LIN {X 0,Y 324.452,Z 606.51,A -85,B 0,C 180,E1 -15849.821,E2 -15849.821} C_VEL
LIN {X 0,Y 327.125,Z 593.397,A -85,B 0,C 180,E1 -15851.148,E2 -15851.148} C_VEL
LIN {X 0,Y 329.681,Z 579.293,A -85,B 0,C 180,E1 -15852.308,E2 -15852.308} C_VEL
LIN {X 0,Y 332.153,Z 563.092,A -85,B 0,C 180,E1 -15853.333,E2 -15853.333} C_VEL
LIN {X 0,Y 333.966,Z 548.09,A -85,B 0,C 180,E1 -15854.029,E2 -15854.029} C_VEL
LIN {X 0,Y 336.479,Z 518.568,A -85,B 0,C 180,E1 -15854.979,E2 -15854.979} C_VEL
LIN {X 0,Y 343.808,Z 437.667,A -85,B 0,C 180,E1 -15857.456,E2 -15857.456} C_VEL
LIN {X 0,Y 343.461,Z 436.268,A -85,B 0,C 180,E1 -15857.604,E2 -15857.604} C_VEL
LIN {X 0,Y 340.27,Z 429.347,A -85,B 0,C 180,E1 -15858.7,E2 -15858.7} C_VEL
LIN {X 0,Y 336.483,Z 422.195,A -85,B 0,C 180,E1 -15860.082,E2 -15860.082} C_VEL
LIN {X 0,Y 332.788,Z 415.874,A -85,B 0,C 180,E1 -15861.56,E2 -15861.56} C_VEL
LIN {X 0,Y 329.389,Z 410.762,A -85,B 0,C 180,E1 -15863.052,E2 -15863.052} C_VEL
LIN {X 0,Y 326.443,Z 406.618,A -85,B 0,C 180,E1 -15864.518,E2 -15864.518} C_VEL
LIN {X 0,Y 322.983,Z 401.962,A -85,B 0,C 180,E1 -15866.589,E2 -15866.589} C_VEL
LIN {X 0,Y 319.205,Z 397.297,A -85,B 0,C 180,E1 -15869.678,E2 -15869.678} C_VEL
LIN {X 0,Y 316.987,Z 395.124,A -85,B 0,C 180,E1 -15872.902,E2 -15872.902} C_VEL
LIN {X 0,Y 316.478,Z 394.789,A -85,B 0,C 180,E1 -15875.266,E2 -15875.266} C_VEL
LIN {X 0,Y 316.828,Z 395.766,A -85,B 0,C 180,E1 -15877.528,E2 -15877.528} C_VEL
LIN {X 0,Y 318.754,Z 398.698,A -85,B 0,C 180,E1 -15880.662,E2 -15880.662} C_VEL
LIN {X 0,Y 320.871,Z 401.495,A -85,B 0,C 180,E1 -15882.648,E2 -15882.648} C_VEL
LIN {X 0,Y 325.084,Z 407.921,A -85,B 0,C 180,E1 -15885.514,E2 -15885.514} C_VEL
LIN {X 0,Y 328.982,Z 414.436,A -85,B 0,C 180,E1 -15887.591,E2 -15887.591} C_VEL
LIN {X 0,Y 332.395,Z 420.455,A -85,B 0,C 180,E1 -15889.134,E2 -15889.134} C_VEL
LIN {X 0,Y 336.259,Z 427.81,A -85,B 0,C 180,E1 -15890.698,E2 -15890.698} C_VEL
LIN {X 0,Y 340.531,Z 437.373,A -85,B 0,C 180,E1 -15892.295,E2 -15892.295} C_VEL
LIN {X 0,Y 342.927,Z 443.986,A -85,B 0,C 180,E1 -15893.182,E2 -15893.182} C_VEL
LIN {X 0,Y 343.146,Z 448.361,A -85,B 0,C 180,E1 -15893.458,E2 -15893.458} C_VEL
LIN {X 0,Y 334.823,Z 544.074,A -85,B 0,C 180,E1 -15896.383,E2 -15896.383} C_VEL
LIN {X 0,Y 333.156,Z 562.468,A -85,B 0,C 180,E1 -15897.006,E2 -15897.006} C_VEL
LIN {X 0,Y 330.94,Z 578.482,A -85,B 0,C 180,E1 -15897.752,E2 -15897.752} C_VEL
LIN {X 0,Y 328.466,Z 592.922,A -85,B 0,C 180,E1 -15898.653,E2 -15898.653} C_VEL
LIN {X 0,Y 325.617,Z 607.581,A -85,B 0,C 180,E1 -15899.828,E2 -15899.828} C_VEL
LIN {X 0,Y 322.66,Z 621.222,A -85,B 0,C 180,E1 -15901.188,E2 -15901.188} C_VEL
LIN {X 0,Y 319.496,Z 634.657,A -85,B 0,C 180,E1 -15902.841,E2 -15902.841} C_VEL
LIN {X 0,Y 316.461,Z 646.925,A -85,B 0,C 180,E1 -15904.689,E2 -15904.689} C_VEL
LIN {X 0,Y 313.386,Z 658.797,A -85,B 0,C 180,E1 -15906.848,E2 -15906.848} C_VEL
LIN {X 0,Y 310.733,Z 669.029,A -85,B 0,C 180,E1 -15909.13,E2 -15909.13} C_VEL
LIN {X 0,Y 308.293,Z 678.544,A -85,B 0,C 180,E1 -15911.731,E2 -15911.731} C_VEL
LIN {X 0,Y 306.546,Z 685.471,A -85,B 0,C 180,E1 -15914.029,E2 -15914.029} C_VEL
LIN {X 0,Y 305.238,Z 691.852,A -85,B 0,C 180,E1 -15916.687,E2 -15916.687} C_VEL
LIN {X 0,Y 304.288,Z 696.815,A -85,B 0,C 180,E1 -15919.35,E2 -15919.35} C_VEL
LIN {X 0,Y 303.795,Z 700.457,A -85,B 0,C 180,E1 -15922.019,E2 -15922.019} C_VEL
LIN {X 0,Y 303.596,Z 702.832,A -85,B 0,C 180,E1 -15924.685,E2 -15924.685} C_VEL
LIN {X 0,Y 303.593,Z 703.983,A -85,B 0,C 180,E1 -15927.344,E2 -15927.344} C_VEL
LIN {X 0,Y 303.605,Z 703.898,A -85,B 0,C 180,E1 -15929.998,E2 -15929.998} C_VEL
LIN {X 0,Y 303.619,Z 702.551,A -85,B 0,C 180,E1 -15932.651,E2 -15932.651} C_VEL
LIN {X 0,Y 303.634,Z 699.89,A -85,B 0,C 180,E1 -15935.31,E2 -15935.31} C_VEL
LIN {X 0,Y 303.805,Z 695.853,A -85,B 0,C 180,E1 -15937.976,E2 -15937.976} C_VEL
LIN {X 0,Y 304.12,Z 690.347,A -85,B 0,C 180,E1 -15940.652,E2 -15940.652} C_VEL
LIN {X 0,Y 304.708,Z 685.156,A -85,B 0,C 180,E1 -15942.655,E2 -15942.655} C_VEL
LIN {X 0,Y 305.549,Z 677.938,A -85,B 0,C 180,E1 -15944.973,E2 -15944.973} C_VEL
LIN {X 0,Y 306.797,Z 669.033,A -85,B 0,C 180,E1 -15947.323,E2 -15947.323} C_VEL
LIN {X 0,Y 308.202,Z 660.042,A -85,B 0,C 180,E1 -15949.306,E2 -15949.306} C_VEL
LIN {X 0,Y 309.836,Z 649.388,A -85,B 0,C 180,E1 -15951.278,E2 -15951.278} C_VEL
LIN {X 0,Y 311.797,Z 636.624,A -85,B 0,C 180,E1 -15953.23,E2 -15953.23} C_VEL
LIN {X 0,Y 313.659,Z 623.857,A -85,B 0,C 180,E1 -15954.84,E2 -15954.84} C_VEL
LIN {X 0,Y 315.546,Z 609.954,A -85,B 0,C 180,E1 -15956.272,E2 -15956.272} C_VEL
LIN {X 0,Y 317.457,Z 594.626,A -85,B 0,C 180,E1 -15957.523,E2 -15957.523} C_VEL
LIN {X 0,Y 319.021,Z 579.208,A -85,B 0,C 180,E1 -15958.492,E2 -15958.492} C_VEL
LIN {X 0,Y 320.355,Z 563.283,A -85,B 0,C 180,E1 -15959.215,E2 -15959.215} C_VEL
LIN {X 0,Y 321.454,Z 541.44,A -85,B 0,C 180,E1 -15959.87,E2 -15959.87} C_VEL
LIN {X 0,Y 325.806,Z 442.848,A -85,B 0,C 180,E1 -15962.583,E2 -15962.583} C_VEL
LIN {X 0,Y 322.744,Z 425.216,A -85,B 0,C 180,E1 -15963.398,E2 -15963.398} C_VEL
LIN {X 0,Y 310.834,Z 396.248,A -85,B 0,C 180,E1 -15965.467,E2 -15965.467} C_VEL
LIN {X 0,Y 309.569,Z 393.101,A -85,B 0,C 180,E1 -15965.719,E2 -15965.719} C_VEL
LIN {X 0,Y 306.644,Z 381.762,A -85,B 0,C 180,E1 -15968.809,E2 -15968.809} C_VEL
LIN {X 0,Y 305.41,Z 377.069,A -85,B 0,C 180,E1 -15970.171,E2 -15970.171} C_VEL
LIN {X 0,Y 305.411,Z 377.066,A -85,B 0,C 180,E1 -15973.654,E2 -15973.654} C_VEL
LIN {X 0,Y 305.424,Z 377.063,A -85,B 0,C 180,E1 -15977.417,E2 -15977.417} C_VEL
LIN {X 0,Y 305.429,Z 377.064,A -85,B 0,C 180,E1 -15981.591,E2 -15981.591} C_VEL
LIN {X 0,Y 305.449,Z 377.06,A -85,B 0,C 180,E1 -15984.885,E2 -15984.885} C_VEL
LIN {X 0,Y 305.429,Z 377.065,A -85,B 0,C 180,E1 -15988.357,E2 -15988.357} C_VEL
LIN {X 0,Y 305.44,Z 377.06,A -85,B 0,C 180,E1 -15991.106,E2 -15991.106} C_VEL
LIN {X 0,Y 305.465,Z 377.06,A -85,B 0,C 180,E1 -15994.079,E2 -15994.079} C_VEL
LIN {X 0,Y 305.447,Z 377.062,A -85,B 0,C 180,E1 -15998.399,E2 -15998.399} C_VEL
LIN {X 0,Y 305.5,Z 377.049,A -85,B 0,C 180,E1 -16001.212,E2 -16001.212} C_VEL
LIN {X 0,Y 305.566,Z 377.045,A -85,B 0,C 180,E1 -16005.345,E2 -16005.345} C_VEL
LIN {X 0,Y 305.609,Z 377.036,A -85,B 0,C 180,E1 -16009.399,E2 -16009.399} C_VEL
LIN {X 0,Y 305.732,Z 377.027,A -85,B 0,C 180,E1 -16012.073,E2 -16012.073} C_VEL
LIN {X 0,Y 305.643,Z 377.035,A -85,B 0,C 180,E1 -16014.723,E2 -16014.723} C_VEL
LIN {X 0,Y 305.92,Z 377.001,A -85,B 0,C 180,E1 -16018.684,E2 -16018.684} C_VEL
LIN {X 0,Y 305.92,Z 377.001,A -85,B 0,C 180,E1 -16021.317,E2 -16021.317} C_VEL
LIN {X 0,Y 305.771,Z 377.02,A -85,B 0,C 180,E1 -16026.6,E2 -16026.6} C_VEL
LIN {X 0,Y 305.68,Z 377.03,A -85,B 0,C 180,E1 -16029.262,E2 -16029.262} C_VEL
LIN {X 0,Y 305.556,Z 377.046,A -85,B 0,C 180,E1 -16033.298,E2 -16033.298} C_VEL
LIN {X 0,Y 305.51,Z 377.051,A -85,B 0,C 180,E1 -16037.401,E2 -16037.401} C_VEL
LIN {X 0,Y 305.468,Z 377.06,A -85,B 0,C 180,E1 -16040.189,E2 -16040.189} C_VEL
LIN {X 0,Y 305.442,Z 377.059,A -85,B 0,C 180,E1 -16044.467,E2 -16044.467} C_VEL
LIN {X 0,Y 305.429,Z 377.061,A -85,B 0,C 180,E1 -16047.401,E2 -16047.401} C_VEL
LIN {X 0,Y 305.406,Z 377.065,A -85,B 0,C 180,E1 -16050.416,E2 -16050.416} C_VEL
LIN {X 0,Y 305.454,Z 377.06,A -85,B 0,C 180,E1 -16054.08,E2 -16054.08} C_VEL
LIN {X 0,Y 305.441,Z 377.059,A -85,B 0,C 180,E1 -16056.745,E2 -16056.745} C_VEL
LIN {X 0,Y 305.4,Z 377.064,A -85,B 0,C 180,E1 -16060.592,E2 -16060.592} C_VEL
LIN {X 0,Y 305.413,Z 377.065,A -85,B 0,C 180,E1 -16063.658,E2 -16063.658} C_VEL
LIN {X 0,Y 305.427,Z 377.064,A -85,B 0,C 180,E1 -16067.421,E2 -16067.421} C_VEL
LIN {X 0,Y 305.435,Z 377.062,A -85,B 0,C 180,E1 -16071.594,E2 -16071.594} C_VEL
LIN {X 0,Y 305.455,Z 377.058,A -85,B 0,C 180,E1 -16074.889,E2 -16074.889} C_VEL
LIN {X 0,Y 305.437,Z 377.06,A -85,B 0,C 180,E1 -16078.361,E2 -16078.361} C_VEL
LIN {X 0,Y 305.45,Z 377.059,A -85,B 0,C 180,E1 -16081.109,E2 -16081.109} C_VEL
LIN {X 0,Y 305.476,Z 377.057,A -85,B 0,C 180,E1 -16084.082,E2 -16084.082} C_VEL
LIN {X 0,Y 305.463,Z 377.058,A -85,B 0,C 180,E1 -16088.403,E2 -16088.403} C_VEL
LIN {X 0,Y 305.542,Z 377.048,A -85,B 0,C 180,E1 -16091.217,E2 -16091.217} C_VEL
LIN {X 0,Y 305.626,Z 377.032,A -85,B 0,C 180,E1 -16095.35,E2 -16095.35} C_VEL
LIN {X 0,Y 305.636,Z 377.038,A -85,B 0,C 180,E1 -16099.402,E2 -16099.402} C_VEL
LIN {X 0,Y 305.747,Z 377.023,A -85,B 0,C 180,E1 -16102.075,E2 -16102.075} C_VEL
LIN {X 0,Y 305.659,Z 377.029,A -85,B 0,C 180,E1 -16104.725,E2 -16104.725} C_VEL
LIN {X 0,Y 305.948,Z 376.997,A -85,B 0,C 180,E1 -16108.686,E2 -16108.686} C_VEL
LIN {X 0,Y 305.939,Z 377.001,A -85,B 0,C 180,E1 -16111.318,E2 -16111.318} C_VEL
LIN {X 0,Y 305.664,Z 377.035,A -85,B 0,C 180,E1 -16115.279,E2 -16115.279} C_VEL
LIN {X 0,Y 305.763,Z 377.022,A -85,B 0,C 180,E1 -16117.929,E2 -16117.929} C_VEL
LIN {X 0,Y 305.6,Z 377.043,A -85,B 0,C 180,E1 -16121.947,E2 -16121.947} C_VEL
LIN {X 0,Y 305.564,Z 377.044,A -85,B 0,C 180,E1 -16124.981,E2 -16124.981} C_VEL
LIN {X 0,Y 305.515,Z 377.05,A -85,B 0,C 180,E1 -16128.789,E2 -16128.789} C_VEL
LIN {X 0,Y 305.492,Z 377.055,A -85,B 0,C 180,E1 -16133.041,E2 -16133.041} C_VEL
LIN {X 0,Y 305.459,Z 377.059,A -85,B 0,C 180,E1 -16136.192,E2 -16136.192} C_VEL
LIN {X 0,Y 305.455,Z 377.061,A -85,B 0,C 180,E1 -16139.035,E2 -16139.035} C_VEL
LIN {X 0,Y 305.443,Z 377.064,A -85,B 0,C 180,E1 -16141.954,E2 -16141.954} C_VEL
LIN {X 0,Y 305.515,Z 377.213,A -85,B 0,C 180,E1 -16145.029,E2 -16145.029} C_VEL
LIN {X 0,Y 306.526,Z 379.933,A -85,B 0,C 180,E1 -16145.226,E2 -16145.226} C_VEL
LIN {X 0,Y 311.318,Z 389.798,A -85,B 0,C 180,E1 -16146.039,E2 -16146.039} C_VEL
LIN {X 0,Y 322.35,Z 415.707,A -85,B 0,C 180,E1 -16147.921,E2 -16147.921} C_VEL
LIN {X 0,Y 326.082,Z 424.987,A -85,B 0,C 180,E1 -16148.538,E2 -16148.538} C_VEL
LIN {X 0,Y 320.68,Z 542.492,A -85,B 0,C 180,E1 -16151.776,E2 -16151.776} C_VEL
LIN {X 0,Y 319.54,Z 558.615,A -85,B 0,C 180,E1 -16152.473,E2 -16152.473} C_VEL
LIN {X 0,Y 318.124,Z 574.349,A -85,B 0,C 180,E1 -16153.424,E2 -16153.424} C_VEL
LIN {X 0,Y 316.452,Z 589.23,A -85,B 0,C 180,E1 -16154.596,E2 -16154.596} C_VEL
LIN {X 0,Y 314.644,Z 603.29,A -85,B 0,C 180,E1 -16155.985,E2 -16155.985} C_VEL
LIN {X 0,Y 312.776,Z 616.701,A -85,B 0,C 180,E1 -16157.616,E2 -16157.616} C_VEL
LIN {X 0,Y 310.867,Z 629.385,A -85,B 0,C 180,E1 -16159.492,E2 -16159.492} C_VEL
LIN {X 0,Y 309.241,Z 639.693,A -85,B 0,C 180,E1 -16161.319,E2 -16161.319} C_VEL
LIN {X 0,Y 307.978,Z 647.89,A -85,B 0,C 180,E1 -16163.009,E2 -16163.009} C_VEL
LIN {X 0,Y 306.745,Z 651.603,A -85,B 0,C 180,E1 -16163.849,E2 -16163.849} C_VEL
LIN {X 0,Y 303.068,Z 657.329,A -85,B 0,C 180,E1 -16165.212,E2 -16165.212} C_VEL
LIN {X 0,Y 299.488,Z 662.573,A -85,B 0,C 180,E1 -16166.655,E2 -16166.655} C_VEL
LIN {X 0,Y 298.416,Z 665.551,A -85,B 0,C 180,E1 -16167.604,E2 -16167.604} C_VEL
LIN {X 0,Y 297.562,Z 672.589,A -85,B 0,C 180,E1 -16170.264,E2 -16170.264} C_VEL
LIN {X 0,Y 297.025,Z 677.318,A -85,B 0,C 180,E1 -16172.522,E2 -16172.522} C_VEL
LIN {X 0,Y 296.632,Z 681.037,A -85,B 0,C 180,E1 -16174.756,E2 -16174.756} C_VEL
LIN {X 0,Y 296.351,Z 684.552,A -85,B 0,C 180,E1 -16177.7,E2 -16177.7} C_VEL
LIN {X 0,Y 296.213,Z 686.564,A -85,B 0,C 180,E1 -16180.599,E2 -16180.599} C_VEL
LIN {X 0,Y 296.266,Z 687.043,A -85,B 0,C 180,E1 -16182.038,E2 -16182.038} C_VEL
LIN {X 0,Y 296.413,Z 686.992,A -85,B 0,C 180,E1 -16184.881,E2 -16184.881} C_VEL
LIN {X 0,Y 296.859,Z 685.634,A -85,B 0,C 180,E1 -16187.697,E2 -16187.697} C_VEL
LIN {X 0,Y 297.577,Z 683.019,A -85,B 0,C 180,E1 -16190.484,E2 -16190.484} C_VEL
LIN {X 0,Y 298.656,Z 679.093,A -85,B 0,C 180,E1 -16193.243,E2 -16193.243} C_VEL
LIN {X 0,Y 300.16,Z 673.803,A -85,B 0,C 180,E1 -16195.972,E2 -16195.972} C_VEL
LIN {X 0,Y 302.276,Z 666.695,A -85,B 0,C 180,E1 -16198.809,E2 -16198.809} C_VEL
LIN {X 0,Y 304.679,Z 658.733,A -85,B 0,C 180,E1 -16201.321,E2 -16201.321} C_VEL
LIN {X 0,Y 307.304,Z 649.837,A -85,B 0,C 180,E1 -16203.605,E2 -16203.605} C_VEL
LIN {X 0,Y 310.461,Z 639.239,A -85,B 0,C 180,E1 -16205.847,E2 -16205.847} C_VEL
LIN {X 0,Y 313.734,Z 627.426,A -85,B 0,C 180,E1 -16207.886,E2 -16207.886} C_VEL
LIN {X 0,Y 317.103,Z 614.32,A -85,B 0,C 180,E1 -16209.729,E2 -16209.729} C_VEL
LIN {X 0,Y 320.152,Z 601.331,A -85,B 0,C 180,E1 -16211.234,E2 -16211.234} C_VEL
LIN {X 0,Y 323.061,Z 587.136,A -85,B 0,C 180,E1 -16212.564,E2 -16212.564} C_VEL
LIN {X 0,Y 325.711,Z 572.302,A -85,B 0,C 180,E1 -16213.651,E2 -16213.651} C_VEL
LIN {X 0,Y 327.75,Z 558.503,A -85,B 0,C 180,E1 -16214.453,E2 -16214.453} C_VEL
LIN {X 0,Y 329.623,Z 542.223,A -85,B 0,C 180,E1 -16215.14,E2 -16215.14} C_VEL
LIN {X 0,Y 339.186,Z 441.013,A -85,B 0,C 180,E1 -16218.308,E2 -16218.308} C_VEL
LIN {X 0,Y 339.127,Z 439.74,A -85,B 0,C 180,E1 -16218.392,E2 -16218.392} C_VEL
LIN {X 0,Y 335.275,Z 431.44,A -85,B 0,C 180,E1 -16219.832,E2 -16219.832} C_VEL
LIN {X 0,Y 331.155,Z 423.968,A -85,B 0,C 180,E1 -16221.494,E2 -16221.494} C_VEL
LIN {X 0,Y 327.497,Z 417.79,A -85,B 0,C 180,E1 -16223.175,E2 -16223.175} C_VEL
LIN {X 0,Y 324.214,Z 413.03,A -85,B 0,C 180,E1 -16224.882,E2 -16224.882} C_VEL
LIN {X 0,Y 321.15,Z 408.709,A -85,B 0,C 180,E1 -16226.809,E2 -16226.809} C_VEL
LIN {X 0,Y 317.586,Z 404.164,A -85,B 0,C 180,E1 -16229.844,E2 -16229.844} C_VEL
LIN {X 0,Y 315.511,Z 402.045,A -85,B 0,C 180,E1 -16232.995,E2 -16232.995} C_VEL
LIN {X 0,Y 315.041,Z 401.783,A -85,B 0,C 180,E1 -16235.451,E2 -16235.451} C_VEL
LIN {X 0,Y 315.502,Z 402.97,A -85,B 0,C 180,E1 -16237.839,E2 -16237.839} C_VEL
LIN {X 0,Y 317.445,Z 406.025,A -85,B 0,C 180,E1 -16240.865,E2 -16240.865} C_VEL
LIN {X 0,Y 319.074,Z 408.27,A -85,B 0,C 180,E1 -16242.403,E2 -16242.403} C_VEL
LIN {X 0,Y 322.847,Z 414.322,A -85,B 0,C 180,E1 -16245.135,E2 -16245.135} C_VEL
LIN {X 0,Y 326.288,Z 420.329,A -85,B 0,C 180,E1 -16247.082,E2 -16247.082} C_VEL
LIN {X 0,Y 329.432,Z 426.175,A -85,B 0,C 180,E1 -16248.617,E2 -16248.617} C_VEL
LIN {X 0,Y 333.083,Z 433.543,A -85,B 0,C 180,E1 -16250.207,E2 -16250.207} C_VEL
LIN {X 0,Y 337.359,Z 443.689,A -85,B 0,C 180,E1 -16251.915,E2 -16251.915} C_VEL
LIN {X 0,Y 338.627,Z 447.338,A -85,B 0,C 180,E1 -16252.402,E2 -16252.402} C_VEL
LIN {X 0,Y 338.62,Z 450.838,A -85,B 0,C 180,E1 -16252.588,E2 -16252.588} C_VEL
LIN {X 0,Y 330.386,Z 539.529,A -85,B 0,C 180,E1 -16255.362,E2 -16255.362} C_VEL
LIN {X 0,Y 328.263,Z 561.131,A -85,B 0,C 180,E1 -16256.081,E2 -16256.081} C_VEL
LIN {X 0,Y 325.98,Z 577.135,A -85,B 0,C 180,E1 -16256.832,E2 -16256.832} C_VEL
LIN {X 0,Y 323.342,Z 591.833,A -85,B 0,C 180,E1 -16257.73,E2 -16257.73} C_VEL
LIN {X 0,Y 320.323,Z 606.661,A -85,B 0,C 180,E1 -16258.916,E2 -16258.916} C_VEL
LIN {X 0,Y 316.915,Z 621.573,A -85,B 0,C 180,E1 -16260.432,E2 -16260.432} C_VEL
LIN {X 0,Y 313.295,Z 635.94,A -85,B 0,C 180,E1 -16262.257,E2 -16262.257} C_VEL
LIN {X 0,Y 310.126,Z 647.958,A -85,B 0,C 180,E1 -16264.134,E2 -16264.134} C_VEL
LIN {X 0,Y 307.304,Z 658.157,A -85,B 0,C 180,E1 -16266.045,E2 -16266.045} C_VEL
LIN {X 0,Y 304.467,Z 668.311,A -85,B 0,C 180,E1 -16268.324,E2 -16268.324} C_VEL
LIN {X 0,Y 302.122,Z 676.804,A -85,B 0,C 180,E1 -16270.639,E2 -16270.639} C_VEL
LIN {X 0,Y 300.204,Z 683.887,A -85,B 0,C 180,E1 -16272.982,E2 -16272.982} C_VEL
LIN {X 0,Y 298.827,Z 689.05,A -85,B 0,C 180,E1 -16275.005,E2 -16275.005} C_VEL
LIN {X 0,Y 297.701,Z 694.624,A -85,B 0,C 180,E1 -16277.731,E2 -16277.731} C_VEL
LIN {X 0,Y 296.951,Z 698.826,A -85,B 0,C 180,E1 -16280.462,E2 -16280.462} C_VEL
LIN {X 0,Y 296.554,Z 701.735,A -85,B 0,C 180,E1 -16283.193,E2 -16283.193} C_VEL
LIN {X 0,Y 296.467,Z 703.408,A -85,B 0,C 180,E1 -16285.92,E2 -16285.92} C_VEL
LIN {X 0,Y 296.491,Z 703.855,A -85,B 0,C 180,E1 -16288.64,E2 -16288.64} C_VEL
LIN {X 0,Y 296.512,Z 703.056,A -85,B 0,C 180,E1 -16291.356,E2 -16291.356} C_VEL
LIN {X 0,Y 296.551,Z 700.983,A -85,B 0,C 180,E1 -16294.075,E2 -16294.075} C_VEL
LIN {X 0,Y 296.629,Z 697.572,A -85,B 0,C 180,E1 -16296.801,E2 -16296.801} C_VEL
LIN {X 0,Y 296.882,Z 692.722,A -85,B 0,C 180,E1 -16299.536,E2 -16299.536} C_VEL
LIN {X 0,Y 297.49,Z 686.32,A -85,B 0,C 180,E1 -16302.274,E2 -16302.274} C_VEL
LIN {X 0,Y 298.239,Z 679.294,A -85,B 0,C 180,E1 -16304.672,E2 -16304.672} C_VEL
LIN {X 0,Y 299.517,Z 670.79,A -85,B 0,C 180,E1 -16307.054,E2 -16307.054} C_VEL
LIN {X 0,Y 301.118,Z 660.526,A -85,B 0,C 180,E1 -16309.424,E2 -16309.424} C_VEL
LIN {X 0,Y 302.819,Z 649.975,A -85,B 0,C 180,E1 -16311.438,E2 -16311.438} C_VEL
LIN {X 0,Y 304.586,Z 638.51,A -85,B 0,C 180,E1 -16313.272,E2 -16313.272} C_VEL
LIN {X 0,Y 306.497,Z 626.146,A -85,B 0,C 180,E1 -16314.917,E2 -16314.917} C_VEL
LIN {X 0,Y 308.403,Z 612.791,A -85,B 0,C 180,E1 -16316.381,E2 -16316.381} C_VEL
LIN {X 0,Y 310.342,Z 598.348,A -85,B 0,C 180,E1 -16317.654,E2 -16317.654} C_VEL
LIN {X 0,Y 311.967,Z 582.868,A -85,B 0,C 180,E1 -16318.728,E2 -16318.728} C_VEL
LIN {X 0,Y 313.407,Z 567.509,A -85,B 0,C 180,E1 -16319.507,E2 -16319.507} C_VEL
LIN {X 0,Y 314.469,Z 550.42,A -85,B 0,C 180,E1 -16320.093,E2 -16320.093} C_VEL
LIN {X 0,Y 319.42,Z 444.085,A -85,B 0,C 180,E1 -16323.081,E2 -16323.081} C_VEL
LIN {X 0,Y 316.595,Z 427.87,A -85,B 0,C 180,E1 -16323.856,E2 -16323.856} C_VEL
LIN {X 0,Y 305.243,Z 399.983,A -85,B 0,C 180,E1 -16325.887,E2 -16325.887} C_VEL
LIN {X 0,Y 302.268,Z 392.932,A -85,B 0,C 180,E1 -16326.455,E2 -16326.455} C_VEL
LIN {X 0,Y 299.308,Z 381.624,A -85,B 0,C 180,E1 -16329.63,E2 -16329.63} C_VEL
LIN {X 0,Y 298.352,Z 377.947,A -85,B 0,C 180,E1 -16330.708,E2 -16330.708} C_VEL
LIN {X 0,Y 298.36,Z 377.944,A -85,B 0,C 180,E1 -16333.096,E2 -16333.096} C_VEL
LIN {X 0,Y 298.36,Z 377.944,A -85,B 0,C 180,E1 -16336.913,E2 -16336.913} C_VEL
LIN {X 0,Y 298.373,Z 377.942,A -85,B 0,C 180,E1 -16341.01,E2 -16341.01} C_VEL
LIN {X 0,Y 298.392,Z 377.943,A -85,B 0,C 180,E1 -16343.927,E2 -16343.927} C_VEL
LIN {X 0,Y 298.38,Z 377.941,A -85,B 0,C 180,E1 -16347.198,E2 -16347.198} C_VEL
LIN {X 0,Y 298.351,Z 377.945,A -85,B 0,C 180,E1 -16350.637,E2 -16350.637} C_VEL
LIN {X 0,Y 298.407,Z 377.935,A -85,B 0,C 180,E1 -16354.917,E2 -16354.917} C_VEL
LIN {X 0,Y 298.403,Z 377.937,A -85,B 0,C 180,E1 -16359.312,E2 -16359.312} C_VEL
LIN {X 0,Y 298.445,Z 377.934,A -85,B 0,C 180,E1 -16362.174,E2 -16362.174} C_VEL
LIN {X 0,Y 298.498,Z 377.925,A -85,B 0,C 180,E1 -16364.99,E2 -16364.99} C_VEL
LIN {X 0,Y 298.568,Z 377.912,A -85,B 0,C 180,E1 -16369.146,E2 -16369.146} C_VEL
LIN {X 0,Y 298.684,Z 377.903,A -85,B 0,C 180,E1 -16371.884,E2 -16371.884} C_VEL
LIN {X 0,Y 298.613,Z 377.912,A -85,B 0,C 180,E1 -16374.598,E2 -16374.598} C_VEL
LIN {X 0,Y 298.888,Z 377.877,A -85,B 0,C 180,E1 -16378.653,E2 -16378.653} C_VEL
LIN {X 0,Y 298.888,Z 377.877,A -85,B 0,C 180,E1 -16381.348,E2 -16381.348} C_VEL
LIN {X 0,Y 298.72,Z 377.898,A -85,B 0,C 180,E1 -16386.756,E2 -16386.756} C_VEL
LIN {X 0,Y 298.611,Z 377.911,A -85,B 0,C 180,E1 -16389.483,E2 -16389.483} C_VEL
LIN {X 0,Y 298.509,Z 377.926,A -85,B 0,C 180,E1 -16393.618,E2 -16393.618} C_VEL
LIN {X 0,Y 298.446,Z 377.931,A -85,B 0,C 180,E1 -16396.415,E2 -16396.415} C_VEL
LIN {X 0,Y 298.427,Z 377.935,A -85,B 0,C 180,E1 -16399.617,E2 -16399.617} C_VEL
LIN {X 0,Y 298.376,Z 377.942,A -85,B 0,C 180,E1 -16403.605,E2 -16403.605} C_VEL
LIN {X 0,Y 298.389,Z 377.937,A -85,B 0,C 180,E1 -16406.584,E2 -16406.584} C_VEL
LIN {X 0,Y 298.346,Z 377.947,A -85,B 0,C 180,E1 -16409.65,E2 -16409.65} C_VEL
LIN {X 0,Y 298.382,Z 377.938,A -85,B 0,C 180,E1 -16412.802,E2 -16412.802} C_VEL
LIN {X 0,Y 298.416,Z 377.934,A -85,B 0,C 180,E1 -16416.804,E2 -16416.804} C_VEL
LIN {X 0,Y 298.364,Z 377.944,A -85,B 0,C 180,E1 -16419.494,E2 -16419.494} C_VEL
LIN {X 0,Y 298.362,Z 377.939,A -85,B 0,C 180,E1 -16423.099,E2 -16423.099} C_VEL
LIN {X 0,Y 298.363,Z 377.942,A -85,B 0,C 180,E1 -16426.917,E2 -16426.917} C_VEL
LIN {X 0,Y 298.344,Z 377.941,A -85,B 0,C 180,E1 -16431.021,E2 -16431.021} C_VEL
LIN {X 0,Y 298.398,Z 377.942,A -85,B 0,C 180,E1 -16433.93,E2 -16433.93} C_VEL
LIN {X 0,Y 298.388,Z 377.939,A -85,B 0,C 180,E1 -16437.202,E2 -16437.202} C_VEL
LIN {X 0,Y 298.36,Z 377.942,A -85,B 0,C 180,E1 -16440.64,E2 -16440.64} C_VEL
LIN {X 0,Y 298.418,Z 377.934,A -85,B 0,C 180,E1 -16444.921,E2 -16444.921} C_VEL
LIN {X 0,Y 298.4,Z 377.942,A -85,B 0,C 180,E1 -16447.865,E2 -16447.865} C_VEL
LIN {X 0,Y 298.502,Z 377.924,A -85,B 0,C 180,E1 -16450.757,E2 -16450.757} C_VEL
LIN {X 0,Y 298.586,Z 377.906,A -85,B 0,C 180,E1 -16454.997,E2 -16454.997} C_VEL
LIN {X 0,Y 298.592,Z 377.914,A -85,B 0,C 180,E1 -16459.149,E2 -16459.149} C_VEL
LIN {X 0,Y 298.699,Z 377.902,A -85,B 0,C 180,E1 -16461.886,E2 -16461.886} C_VEL
LIN {X 0,Y 298.629,Z 377.904,A -85,B 0,C 180,E1 -16464.6,E2 -16464.6} C_VEL
LIN {X 0,Y 298.915,Z 377.874,A -85,B 0,C 180,E1 -16468.655,E2 -16468.655} C_VEL
LIN {X 0,Y 298.906,Z 377.877,A -85,B 0,C 180,E1 -16471.349,E2 -16471.349} C_VEL
LIN {X 0,Y 298.744,Z 377.896,A -85,B 0,C 180,E1 -16476.757,E2 -16476.757} C_VEL
LIN {X 0,Y 298.63,Z 377.911,A -85,B 0,C 180,E1 -16479.484,E2 -16479.484} C_VEL
LIN {X 0,Y 298.529,Z 377.924,A -85,B 0,C 180,E1 -16483.618,E2 -16483.618} C_VEL
LIN {X 0,Y 298.46,Z 377.93,A -85,B 0,C 180,E1 -16486.416,E2 -16486.416} C_VEL
LIN {X 0,Y 298.464,Z 377.934,A -85,B 0,C 180,E1 -16489.628,E2 -16489.628} C_VEL
LIN {X 0,Y 298.422,Z 377.94,A -85,B 0,C 180,E1 -16493.603,E2 -16493.603} C_VEL
LIN {X 0,Y 298.409,Z 377.937,A -85,B 0,C 180,E1 -16496.584,E2 -16496.584} C_VEL
LIN {X 0,Y 298.4,Z 377.942,A -85,B 0,C 180,E1 -16499.645,E2 -16499.645} C_VEL
LIN {X 0,Y 298.442,Z 377.937,A -85,B 0,C 180,E1 -16504.009,E2 -16504.009} C_VEL
LIN {X 0,Y 298.437,Z 377.936,A -85,B 0,C 180,E1 -16504.315,E2 -16504.315} C_VEL
LIN {X 0,Y 299.471,Z 380.811,A -85,B 0,C 180,E1 -16504.536,E2 -16504.536} C_VEL
LIN {X 0,Y 305.256,Z 392.555,A -85,B 0,C 180,E1 -16505.547,E2 -16505.547} C_VEL
LIN {X 0,Y 316.025,Z 417.81,A -85,B 0,C 180,E1 -16507.425,E2 -16507.425} C_VEL
LIN {X 0,Y 319.644,Z 426.763,A -85,B 0,C 180,E1 -16508.04,E2 -16508.04} C_VEL
LIN {X 0,Y 314.082,Z 542.928,A -85,B 0,C 180,E1 -16511.322,E2 -16511.322} C_VEL
LIN {X 0,Y 312.92,Z 558.734,A -85,B 0,C 180,E1 -16512.019,E2 -16512.019} C_VEL
LIN {X 0,Y 311.501,Z 574.104,A -85,B 0,C 180,E1 -16512.963,E2 -16512.963} C_VEL
LIN {X 0,Y 309.761,Z 589.124,A -85,B 0,C 180,E1 -16514.162,E2 -16514.162} C_VEL
LIN {X 0,Y 307.816,Z 603.741,A -85,B 0,C 180,E1 -16515.635,E2 -16515.635} C_VEL
LIN {X 0,Y 305.858,Z 617.372,A -85,B 0,C 180,E1 -16517.334,E2 -16517.334} C_VEL
LIN {X 0,Y 303.949,Z 629.768,A -85,B 0,C 180,E1 -16519.216,E2 -16519.216} C_VEL
LIN {X 0,Y 302.258,Z 640.203,A -85,B 0,C 180,E1 -16521.112,E2 -16521.112} C_VEL
LIN {X 0,Y 300.611,Z 650.718,A -85,B 0,C 180,E1 -16523.404,E2 -16523.404} C_VEL
LIN {X 0,Y 299.259,Z 659.412,A -85,B 0,C 180,E1 -16525.692,E2 -16525.692} C_VEL
LIN {X 0,Y 298.416,Z 665.551,A -85,B 0,C 180,E1 -16527.604,E2 -16527.604} C_VEL
LIN {X 0,Y 297.377,Z 668.411,A -85,B 0,C 180,E1 -16528.578,E2 -16528.578} C_VEL
LIN {X 0,Y 293.991,Z 672.622,A -85,B 0,C 180,E1 -16530.191,E2 -16530.191} C_VEL
LIN {X 0,Y 290.711,Z 676.311,A -85,B 0,C 180,E1 -16531.887,E2 -16531.887} C_VEL
LIN {X 0,Y 289.862,Z 678.327,A -85,B 0,C 180,E1 -16532.975,E2 -16532.975} C_VEL
LIN {X 0,Y 289.384,Z 682.358,A -85,B 0,C 180,E1 -16535.615,E2 -16535.615} C_VEL
LIN {X 0,Y 289.26,Z 684.409,A -85,B 0,C 180,E1 -16537.412,E2 -16537.412} C_VEL
LIN {X 0,Y 289.133,Z 686.47,A -85,B 0,C 180,E1 -16540.104,E2 -16540.104} C_VEL
LIN {X 0,Y 289.19,Z 687.4,A -85,B 0,C 180,E1 -16543.044,E2 -16543.044} C_VEL
LIN {X 0,Y 289.516,Z 686.916,A -85,B 0,C 180,E1 -16546.173,E2 -16546.173} C_VEL
LIN {X 0,Y 290.01,Z 685.293,A -85,B 0,C 180,E1 -16548.821,E2 -16548.821} C_VEL
LIN {X 0,Y 291.035,Z 681.984,A -85,B 0,C 180,E1 -16551.932,E2 -16551.932} C_VEL
LIN {X 0,Y 292.188,Z 678.07,A -85,B 0,C 180,E1 -16554.479,E2 -16554.479} C_VEL
LIN {X 0,Y 293.983,Z 672.461,A -85,B 0,C 180,E1 -16557.259,E2 -16557.259} C_VEL
LIN {X 0,Y 296.247,Z 665.349,A -85,B 0,C 180,E1 -16560,E2 -16560} C_VEL
LIN {X 0,Y 299.086,Z 656.561,A -85,B 0,C 180,E1 -16562.693,E2 -16562.693} C_VEL
LIN {X 0,Y 302.085,Z 647.247,A -85,B 0,C 180,E1 -16565.005,E2 -16565.005} C_VEL
LIN {X 0,Y 305.474,Z 636.234,A -85,B 0,C 180,E1 -16567.234,E2 -16567.234} C_VEL
LIN {X 0,Y 308.843,Z 624.704,A -85,B 0,C 180,E1 -16569.165,E2 -16569.165} C_VEL
LIN {X 0,Y 312.156,Z 612.34,A -85,B 0,C 180,E1 -16570.868,E2 -16570.868} C_VEL
LIN {X 0,Y 315.459,Z 598.809,A -85,B 0,C 180,E1 -16572.382,E2 -16572.382} C_VEL
LIN {X 0,Y 318.168,Z 586.129,A -85,B 0,C 180,E1 -16573.557,E2 -16573.557} C_VEL
LIN {X 0,Y 321.001,Z 570.965,A -85,B 0,C 180,E1 -16574.665,E2 -16574.665} C_VEL
LIN {X 0,Y 323.31,Z 555.555,A -85,B 0,C 180,E1 -16575.524,E2 -16575.524} C_VEL
LIN {X 0,Y 325.279,Z 538.493,A -85,B 0,C 180,E1 -16576.191,E2 -16576.191} C_VEL
LIN {X 0,Y 334.765,Z 444.063,A -85,B 0,C 180,E1 -16579.206,E2 -16579.206} C_VEL
LIN {X 0,Y 334.731,Z 442.837,A -85,B 0,C 180,E1 -16579.287,E2 -16579.287} C_VEL
LIN {X 0,Y 330.67,Z 434.216,A -85,B 0,C 180,E1 -16580.933,E2 -16580.933} C_VEL
LIN {X 0,Y 326.849,Z 427.251,A -85,B 0,C 180,E1 -16582.646,E2 -16582.646} C_VEL
LIN {X 0,Y 324.275,Z 423.039,A -85,B 0,C 180,E1 -16583.936,E2 -16583.936} C_VEL
LIN {X 0,Y 321.87,Z 419.311,A -85,B 0,C 180,E1 -16585.314,E2 -16585.314} C_VEL
LIN {X 0,Y 319.167,Z 415.297,A -85,B 0,C 180,E1 -16587.136,E2 -16587.136} C_VEL
LIN {X 0,Y 315.978,Z 411.027,A -85,B 0,C 180,E1 -16590.012,E2 -16590.012} C_VEL
LIN {X 0,Y 314,Z 408.924,A -85,B 0,C 180,E1 -16593.174,E2 -16593.174} C_VEL
LIN {X 0,Y 313.656,Z 408.808,A -85,B 0,C 180,E1 -16595.929,E2 -16595.929} C_VEL
LIN {X 0,Y 314.451,Z 410.753,A -85,B 0,C 180,E1 -16598.741,E2 -16598.741} C_VEL
LIN {X 0,Y 316.851,Z 414.176,A -85,B 0,C 180,E1 -16601.714,E2 -16601.714} C_VEL
LIN {X 0,Y 320.66,Z 420.804,A -85,B 0,C 180,E1 -16604.774,E2 -16604.774} C_VEL
LIN {X 0,Y 323.864,Z 426.734,A -85,B 0,C 180,E1 -16606.707,E2 -16606.707} C_VEL
LIN {X 0,Y 326.571,Z 431.988,A -85,B 0,C 180,E1 -16608.111,E2 -16608.111} C_VEL
LIN {X 0,Y 329.931,Z 439.147,A -85,B 0,C 180,E1 -16609.668,E2 -16609.668} C_VEL
LIN {X 0,Y 333.796,Z 448.773,A -85,B 0,C 180,E1 -16611.318,E2 -16611.318} C_VEL
LIN {X 0,Y 334.441,Z 450.771,A -85,B 0,C 180,E1 -16611.603,E2 -16611.603} C_VEL
LIN {X 0,Y 323.578,Z 559.492,A -85,B 0,C 180,E1 -16615.096,E2 -16615.096} C_VEL
LIN {X 0,Y 321.137,Z 576.408,A -85,B 0,C 180,E1 -16615.887,E2 -16615.887} C_VEL
LIN {X 0,Y 318.18,Z 592.007,A -85,B 0,C 180,E1 -16616.859,E2 -16616.859} C_VEL
LIN {X 0,Y 314.95,Z 606.819,A -85,B 0,C 180,E1 -16618.072,E2 -16618.072} C_VEL
LIN {X 0,Y 311.614,Z 620.769,A -85,B 0,C 180,E1 -16619.504,E2 -16619.504} C_VEL
LIN {X 0,Y 308.127,Z 634.068,A -85,B 0,C 180,E1 -16621.193,E2 -16621.193} C_VEL
LIN {X 0,Y 304.987,Z 645.262,A -85,B 0,C 180,E1 -16622.926,E2 -16622.926} C_VEL
LIN {X 0,Y 301.874,Z 655.828,A -85,B 0,C 180,E1 -16624.855,E2 -16624.855} C_VEL
LIN {X 0,Y 299.077,Z 664.879,A -85,B 0,C 180,E1 -16626.819,E2 -16626.819} C_VEL
LIN {X 0,Y 296.414,Z 673.846,A -85,B 0,C 180,E1 -16629.165,E2 -16629.165} C_VEL
LIN {X 0,Y 294.535,Z 680.426,A -85,B 0,C 180,E1 -16631.206,E2 -16631.206} C_VEL
LIN {X 0,Y 292.383,Z 687.579,A -85,B 0,C 180,E1 -16633.895,E2 -16633.895} C_VEL
LIN {X 0,Y 291.05,Z 693.482,A -85,B 0,C 180,E1 -16636.736,E2 -16636.736} C_VEL
LIN {X 0,Y 290.223,Z 696.951,A -85,B 0,C 180,E1 -16638.828,E2 -16638.828} C_VEL
LIN {X 0,Y 289.664,Z 700.433,A -85,B 0,C 180,E1 -16641.627,E2 -16641.627} C_VEL
LIN {X 0,Y 289.427,Z 702.742,A -85,B 0,C 180,E1 -16644.609,E2 -16644.609} C_VEL
LIN {X 0,Y 289.419,Z 703.593,A -85,B 0,C 180,E1 -16647.214,E2 -16647.214} C_VEL
LIN {X 0,Y 289.438,Z 703.326,A -85,B 0,C 180,E1 -16649.998,E2 -16649.998} C_VEL
LIN {X 0,Y 289.471,Z 701.796,A -85,B 0,C 180,E1 -16652.781,E2 -16652.781} C_VEL
LIN {X 0,Y 289.499,Z 698.958,A -85,B 0,C 180,E1 -16655.57,E2 -16655.57} C_VEL
LIN {X 0,Y 289.68,Z 694.738,A -85,B 0,C 180,E1 -16658.368,E2 -16658.368} C_VEL
LIN {X 0,Y 290.047,Z 689.008,A -85,B 0,C 180,E1 -16661.175,E2 -16661.175} C_VEL
LIN {X 0,Y 290.822,Z 682.687,A -85,B 0,C 180,E1 -16663.626,E2 -16663.626} C_VEL
LIN {X 0,Y 291.88,Z 674.925,A -85,B 0,C 180,E1 -16666.073,E2 -16666.073} C_VEL
LIN {X 0,Y 293.256,Z 665.539,A -85,B 0,C 180,E1 -16668.512,E2 -16668.512} C_VEL
LIN {X 0,Y 294.87,Z 655.932,A -85,B 0,C 180,E1 -16670.58,E2 -16670.58} C_VEL
LIN {X 0,Y 296.645,Z 644.754,A -85,B 0,C 180,E1 -16672.603,E2 -16672.603} C_VEL
LIN {X 0,Y 298.525,Z 633.332,A -85,B 0,C 180,E1 -16674.328,E2 -16674.328} C_VEL
LIN {X 0,Y 300.592,Z 619.993,A -85,B 0,C 180,E1 -16675.998,E2 -16675.998} C_VEL
LIN {X 0,Y 302.632,Z 605.349,A -85,B 0,C 180,E1 -16677.485,E2 -16677.485} C_VEL
LIN {X 0,Y 304.557,Z 590.331,A -85,B 0,C 180,E1 -16678.683,E2 -16678.683} C_VEL
LIN {X 0,Y 306.081,Z 575.704,A -85,B 0,C 180,E1 -16679.579,E2 -16679.579} C_VEL
LIN {X 0,Y 307.379,Z 559.601,A -85,B 0,C 180,E1 -16680.292,E2 -16680.292} C_VEL
LIN {X 0,Y 312.947,Z 444.922,A -85,B 0,C 180,E1 -16683.622,E2 -16683.622} C_VEL
LIN {X 0,Y 310.521,Z 430.46,A -85,B 0,C 180,E1 -16684.331,E2 -16684.331} C_VEL
LIN {X 0,Y 298.148,Z 400.247,A -85,B 0,C 180,E1 -16686.588,E2 -16686.588} C_VEL
LIN {X 0,Y 294.969,Z 392.699,A -85,B 0,C 180,E1 -16687.231,E2 -16687.231} C_VEL
LIN {X 0,Y 291.301,Z 378.825,A -85,B 0,C 180,E1 -16691.325,E2 -16691.325} C_VEL
LIN {X 0,Y 291.271,Z 378.827,A -85,B 0,C 180,E1 -16695.595,E2 -16695.595} C_VEL
LIN {X 0,Y 291.288,Z 378.825,A -85,B 0,C 180,E1 -16699.35,E2 -16699.35} C_VEL
LIN {X 0,Y 291.373,Z 378.814,A -85,B 0,C 180,E1 -16702.915,E2 -16702.915} C_VEL
LIN {X 0,Y 291.331,Z 378.823,A -85,B 0,C 180,E1 -16706.3,E2 -16706.3} C_VEL
LIN {X 0,Y 291.322,Z 378.823,A -85,B 0,C 180,E1 -16710.277,E2 -16710.277} C_VEL
LIN {X 0,Y 291.332,Z 378.819,A -85,B 0,C 180,E1 -16714.264,E2 -16714.264} C_VEL
LIN {X 0,Y 291.337,Z 378.818,A -85,B 0,C 180,E1 -16717.296,E2 -16717.296} C_VEL
LIN {X 0,Y 291.373,Z 378.812,A -85,B 0,C 180,E1 -16720.265,E2 -16720.265} C_VEL
LIN {X 0,Y 291.46,Z 378.803,A -85,B 0,C 180,E1 -16724.682,E2 -16724.682} C_VEL
LIN {X 0,Y 291.513,Z 378.79,A -85,B 0,C 180,E1 -16728.88,E2 -16728.88} C_VEL
LIN {X 0,Y 291.637,Z 378.779,A -85,B 0,C 180,E1 -16731.687,E2 -16731.687} C_VEL
LIN {X 0,Y 291.583,Z 378.788,A -85,B 0,C 180,E1 -16734.468,E2 -16734.468} C_VEL
LIN {X 0,Y 291.856,Z 378.753,A -85,B 0,C 180,E1 -16738.621,E2 -16738.621} C_VEL
LIN {X 0,Y 291.855,Z 378.753,A -85,B 0,C 180,E1 -16741.38,E2 -16741.38} C_VEL
LIN {X 0,Y 291.673,Z 378.775,A -85,B 0,C 180,E1 -16746.92,E2 -16746.92} C_VEL
LIN {X 0,Y 291.554,Z 378.792,A -85,B 0,C 180,E1 -16749.715,E2 -16749.715} C_VEL
LIN {X 0,Y 291.468,Z 378.806,A -85,B 0,C 180,E1 -16753.953,E2 -16753.953} C_VEL
LIN {X 0,Y 291.382,Z 378.812,A -85,B 0,C 180,E1 -16758.274,E2 -16758.274} C_VEL
LIN {X 0,Y 291.332,Z 378.818,A -85,B 0,C 180,E1 -16761.215,E2 -16761.215} C_VEL
LIN {X 0,Y 291.321,Z 378.819,A -85,B 0,C 180,E1 -16764.213,E2 -16764.213} C_VEL
LIN {X 0,Y 291.317,Z 378.818,A -85,B 0,C 180,E1 -16767.283,E2 -16767.283} C_VEL
LIN {X 0,Y 291.291,Z 378.824,A -85,B 0,C 180,E1 -16770.443,E2 -16770.443} C_VEL
LIN {X 0,Y 291.333,Z 378.819,A -85,B 0,C 180,E1 -16773.7,E2 -16773.7} C_VEL
LIN {X 0,Y 291.342,Z 378.816,A -85,B 0,C 180,E1 -16777.25,E2 -16777.25} C_VEL
LIN {X 0,Y 291.291,Z 378.821,A -85,B 0,C 180,E1 -16780.65,E2 -16780.65} C_VEL
LIN {X 0,Y 291.274,Z 378.825,A -85,B 0,C 180,E1 -16784.406,E2 -16784.406} C_VEL
LIN {X 0,Y 291.287,Z 378.823,A -85,B 0,C 180,E1 -16788.414,E2 -16788.414} C_VEL
LIN {X 0,Y 291.379,Z 378.811,A -85,B 0,C 180,E1 -16792.918,E2 -16792.918} C_VEL
LIN {X 0,Y 291.338,Z 378.817,A -85,B 0,C 180,E1 -16796.304,E2 -16796.304} C_VEL
LIN {X 0,Y 291.331,Z 378.819,A -85,B 0,C 180,E1 -16800.281,E2 -16800.281} C_VEL
LIN {X 0,Y 291.343,Z 378.816,A -85,B 0,C 180,E1 -16804.268,E2 -16804.268} C_VEL
LIN {X 0,Y 291.357,Z 378.815,A -85,B 0,C 180,E1 -16807.3,E2 -16807.3} C_VEL
LIN {X 0,Y 291.438,Z 378.805,A -85,B 0,C 180,E1 -16810.271,E2 -16810.271} C_VEL
LIN {X 0,Y 291.497,Z 378.787,A -85,B 0,C 180,E1 -16814.668,E2 -16814.668} C_VEL
LIN {X 0,Y 291.536,Z 378.792,A -85,B 0,C 180,E1 -16818.883,E2 -16818.883} C_VEL
LIN {X 0,Y 291.653,Z 378.782,A -85,B 0,C 180,E1 -16821.689,E2 -16821.689} C_VEL
LIN {X 0,Y 291.599,Z 378.779,A -85,B 0,C 180,E1 -16824.47,E2 -16824.47} C_VEL
LIN {X 0,Y 291.881,Z 378.75,A -85,B 0,C 180,E1 -16828.622,E2 -16828.622} C_VEL
LIN {X 0,Y 291.874,Z 378.753,A -85,B 0,C 180,E1 -16831.382,E2 -16831.382} C_VEL
LIN {X 0,Y 291.696,Z 378.774,A -85,B 0,C 180,E1 -16836.921,E2 -16836.921} C_VEL
LIN {X 0,Y 291.573,Z 378.79,A -85,B 0,C 180,E1 -16839.716,E2 -16839.716} C_VEL
LIN {X 0,Y 291.487,Z 378.799,A -85,B 0,C 180,E1 -16843.954,E2 -16843.954} C_VEL
LIN {X 0,Y 291.398,Z 378.809,A -85,B 0,C 180,E1 -16848.274,E2 -16848.274} C_VEL
LIN {X 0,Y 291.366,Z 378.817,A -85,B 0,C 180,E1 -16851.214,E2 -16851.214} C_VEL
LIN {X 0,Y 291.356,Z 378.816,A -85,B 0,C 180,E1 -16854.211,E2 -16854.211} C_VEL
LIN {X 0,Y 291.357,Z 378.818,A -85,B 0,C 180,E1 -16857.28,E2 -16857.28} C_VEL
LIN {X 0,Y 291.325,Z 378.821,A -85,B 0,C 180,E1 -16860.44,E2 -16860.44} C_VEL
LIN {X 0,Y 291.414,Z 378.834,A -85,B 0,C 180,E1 -16863.602,E2 -16863.602} C_VEL
LIN {X 0,Y 292.397,Z 381.656,A -85,B 0,C 180,E1 -16863.814,E2 -16863.814} C_VEL
LIN {X 0,Y 299.127,Z 395.138,A -85,B 0,C 180,E1 -16865.023,E2 -16865.023} C_VEL
LIN {X 0,Y 309.326,Z 418.968,A -85,B 0,C 180,E1 -16866.843,E2 -16866.843} C_VEL
LIN {X 0,Y 313.243,Z 428.722,A -85,B 0,C 180,E1 -16867.531,E2 -16867.531} C_VEL
LIN {X 0,Y 307.483,Z 543.32,A -85,B 0,C 180,E1 -16870.851,E2 -16870.851} C_VEL
LIN {X 0,Y 306.285,Z 559.008,A -85,B 0,C 180,E1 -16871.562,E2 -16871.562} C_VEL
LIN {X 0,Y 304.891,Z 573.582,A -85,B 0,C 180,E1 -16872.47,E2 -16872.47} C_VEL
LIN {X 0,Y 303.292,Z 587.71,A -85,B 0,C 180,E1 -16873.602,E2 -16873.602} C_VEL
LIN {X 0,Y 301.466,Z 600.996,A -85,B 0,C 180,E1 -16874.917,E2 -16874.917} C_VEL
LIN {X 0,Y 299.564,Z 614.169,A -85,B 0,C 180,E1 -16876.517,E2 -16876.517} C_VEL
LIN {X 0,Y 297.547,Z 626.745,A -85,B 0,C 180,E1 -16878.37,E2 -16878.37} C_VEL
LIN {X 0,Y 295.911,Z 636.668,A -85,B 0,C 180,E1 -16880.114,E2 -16880.114} C_VEL
LIN {X 0,Y 294.094,Z 647.86,A -85,B 0,C 180,E1 -16882.455,E2 -16882.455} C_VEL
LIN {X 0,Y 292.639,Z 657.096,A -85,B 0,C 180,E1 -16884.803,E2 -16884.803} C_VEL
LIN {X 0,Y 291.298,Z 666.101,A -85,B 0,C 180,E1 -16887.613,E2 -16887.613} C_VEL
LIN {X 0,Y 290.499,Z 672.569,A -85,B 0,C 180,E1 -16890.116,E2 -16890.116} C_VEL
LIN {X 0,Y 289.862,Z 678.327,A -85,B 0,C 180,E1 -16892.975,E2 -16892.975} C_VEL
LIN {X 0,Y 289.029,Z 680.185,A -85,B 0,C 180,E1 -16894.073,E2 -16894.073} C_VEL
LIN {X 0,Y 285.881,Z 682.761,A -85,B 0,C 180,E1 -16895.876,E2 -16895.876} C_VEL
LIN {X 0,Y 283.266,Z 684.451,A -85,B 0,C 180,E1 -16897.362,E2 -16897.362} C_VEL
LIN {X 0,Y 282.134,Z 685.483,A -85,B 0,C 180,E1 -16898.528,E2 -16898.528} C_VEL
LIN {X 0,Y 282.033,Z 685.74,A -85,B 0,C 180,E1 -16898.926,E2 -16898.926} C_VEL
LIN {X 0,Y 282.044,Z 687.107,A -85,B 0,C 180,E1 -16901.247,E2 -16901.247} C_VEL
LIN {X 0,Y 282.141,Z 687.637,A -85,B 0,C 180,E1 -16904.097,E2 -16904.097} C_VEL
LIN {X 0,Y 282.551,Z 686.908,A -85,B 0,C 180,E1 -16907.064,E2 -16907.064} C_VEL
LIN {X 0,Y 283.257,Z 684.906,A -85,B 0,C 180,E1 -16909.998,E2 -16909.998} C_VEL
LIN {X 0,Y 284.368,Z 681.651,A -85,B 0,C 180,E1 -16912.901,E2 -16912.901} C_VEL
LIN {X 0,Y 285.898,Z 677.074,A -85,B 0,C 180,E1 -16915.77,E2 -16915.77} C_VEL
LIN {X 0,Y 287.966,Z 671.089,A -85,B 0,C 180,E1 -16918.601,E2 -16918.601} C_VEL
LIN {X 0,Y 290.53,Z 663.649,A -85,B 0,C 180,E1 -16921.386,E2 -16921.386} C_VEL
LIN {X 0,Y 293.379,Z 655.624,A -85,B 0,C 180,E1 -16923.777,E2 -16923.777} C_VEL
LIN {X 0,Y 296.666,Z 645.835,A -85,B 0,C 180,E1 -16926.188,E2 -16926.188} C_VEL
LIN {X 0,Y 300.304,Z 634.762,A -85,B 0,C 180,E1 -16928.41,E2 -16928.41} C_VEL
LIN {X 0,Y 304.199,Z 621.971,A -85,B 0,C 180,E1 -16930.482,E2 -16930.482} C_VEL
LIN {X 0,Y 307.803,Z 609.112,A -85,B 0,C 180,E1 -16932.193,E2 -16932.193} C_VEL
LIN {X 0,Y 311.166,Z 595.688,A -85,B 0,C 180,E1 -16933.643,E2 -16933.643} C_VEL
LIN {X 0,Y 314.018,Z 582.388,A -85,B 0,C 180,E1 -16934.816,E2 -16934.816} C_VEL
LIN {X 0,Y 317.033,Z 566.25,A -85,B 0,C 180,E1 -16935.922,E2 -16935.922} C_VEL
LIN {X 0,Y 319.362,Z 550.788,A -85,B 0,C 180,E1 -16936.706,E2 -16936.706} C_VEL
LIN {X 0,Y 321.522,Z 530.982,A -85,B 0,C 180,E1 -16937.409,E2 -16937.409} C_VEL
LIN {X 0,Y 330.566,Z 446.377,A -85,B 0,C 180,E1 -16940.165,E2 -16940.165} C_VEL
LIN {X 0,Y 327.135,Z 438.934,A -85,B 0,C 180,E1 -16941.683,E2 -16941.683} C_VEL
LIN {X 0,Y 323.809,Z 432.663,A -85,B 0,C 180,E1 -16943.305,E2 -16943.305} C_VEL
LIN {X 0,Y 321.544,Z 428.77,A -85,B 0,C 180,E1 -16944.537,E2 -16944.537} C_VEL
LIN {X 0,Y 319.323,Z 425.294,A -85,B 0,C 180,E1 -16945.879,E2 -16945.879} C_VEL
LIN {X 0,Y 317.06,Z 421.744,A -85,B 0,C 180,E1 -16947.543,E2 -16947.543} C_VEL
LIN {X 0,Y 314.372,Z 417.887,A -85,B 0,C 180,E1 -16950.181,E2 -16950.181} C_VEL
LIN {X 0,Y 312.491,Z 415.809,A -85,B 0,C 180,E1 -16953.355,E2 -16953.355} C_VEL
LIN {X 0,Y 312.23,Z 415.901,A -85,B 0,C 180,E1 -16956.119,E2 -16956.119} C_VEL
LIN {X 0,Y 313.039,Z 417.834,A -85,B 0,C 180,E1 -16958.818,E2 -16958.818} C_VEL
LIN {X 0,Y 315.181,Z 421.09,A -85,B 0,C 180,E1 -16961.556,E2 -16961.556} C_VEL
LIN {X 0,Y 318.499,Z 427.226,A -85,B 0,C 180,E1 -16964.386,E2 -16964.386} C_VEL
LIN {X 0,Y 321.299,Z 432.715,A -85,B 0,C 180,E1 -16966.206,E2 -16966.206} C_VEL
LIN {X 0,Y 324.118,Z 438.551,A -85,B 0,C 180,E1 -16967.762,E2 -16967.762} C_VEL
LIN {X 0,Y 327.228,Z 445.717,A -85,B 0,C 180,E1 -16969.303,E2 -16969.303} C_VEL
LIN {X 0,Y 330.159,Z 453.574,A -85,B 0,C 180,E1 -16970.666,E2 -16970.666} C_VEL
LIN {X 0,Y 320.515,Z 545.513,A -85,B 0,C 180,E1 -16973.648,E2 -16973.648} C_VEL
LIN {X 0,Y 318.447,Z 563.342,A -85,B 0,C 180,E1 -16974.304,E2 -16974.304} C_VEL
LIN {X 0,Y 315.718,Z 579.583,A -85,B 0,C 180,E1 -16975.121,E2 -16975.121} C_VEL
LIN {X 0,Y 312.421,Z 595.596,A -85,B 0,C 180,E1 -16976.205,E2 -16976.205} C_VEL
LIN {X 0,Y 309.174,Z 609.393,A -85,B 0,C 180,E1 -16977.403,E2 -16977.403} C_VEL
LIN {X 0,Y 305.667,Z 622.72,A -85,B 0,C 180,E1 -16978.845,E2 -16978.845} C_VEL
LIN {X 0,Y 301.703,Z 636.634,A -85,B 0,C 180,E1 -16980.711,E2 -16980.711} C_VEL
LIN {X 0,Y 298.187,Z 648.369,A -85,B 0,C 180,E1 -16982.637,E2 -16982.637} C_VEL
LIN {X 0,Y 295.006,Z 658.38,A -85,B 0,C 180,E1 -16984.606,E2 -16984.606} C_VEL
LIN {X 0,Y 291.795,Z 668.346,A -85,B 0,C 180,E1 -16986.957,E2 -16986.957} C_VEL
LIN {X 0,Y 289.138,Z 676.731,A -85,B 0,C 180,E1 -16989.361,E2 -16989.361} C_VEL
LIN {X 0,Y 286.61,Z 684.648,A -85,B 0,C 180,E1 -16992.149,E2 -16992.149} C_VEL
LIN {X 0,Y 284.673,Z 691.041,A -85,B 0,C 180,E1 -16994.974,E2 -16994.974} C_VEL
LIN {X 0,Y 283.491,Z 695.994,A -85,B 0,C 180,E1 -16997.833,E2 -16997.833} C_VEL
LIN {X 0,Y 282.861,Z 698.859,A -85,B 0,C 180,E1 -16999.982,E2 -16999.982} C_VEL
LIN {X 0,Y 282.396,Z 701.621,A -85,B 0,C 180,E1 -17002.85,E2 -17002.85} C_VEL
LIN {X 0,Y 282.283,Z 703.118,A -85,B 0,C 180,E1 -17005.714,E2 -17005.714} C_VEL
LIN {X 0,Y 282.335,Z 703.374,A -85,B 0,C 180,E1 -17008.572,E2 -17008.572} C_VEL
LIN {X 0,Y 282.355,Z 702.383,A -85,B 0,C 180,E1 -17011.424,E2 -17011.424} C_VEL
LIN {X 0,Y 282.399,Z 701.41,A -85,B 0,C 180,E1 -17012.851,E2 -17012.851} C_VEL
LIN {X 0,Y 282.409,Z 698.463,A -85,B 0,C 180,E1 -17015.711,E2 -17015.711} C_VEL
LIN {X 0,Y 282.605,Z 694.126,A -85,B 0,C 180,E1 -17018.579,E2 -17018.579} C_VEL
LIN {X 0,Y 283.019,Z 688.267,A -85,B 0,C 180,E1 -17021.456,E2 -17021.456} C_VEL
LIN {X 0,Y 283.842,Z 681.811,A -85,B 0,C 180,E1 -17023.968,E2 -17023.968} C_VEL
LIN {X 0,Y 284.935,Z 673.918,A -85,B 0,C 180,E1 -17026.476,E2 -17026.476} C_VEL
LIN {X 0,Y 286.414,Z 664.347,A -85,B 0,C 180,E1 -17028.971,E2 -17028.971} C_VEL
LIN {X 0,Y 288.087,Z 654.589,A -85,B 0,C 180,E1 -17031.087,E2 -17031.087} C_VEL
LIN {X 0,Y 290.01,Z 642.978,A -85,B 0,C 180,E1 -17033.188,E2 -17033.188} C_VEL
LIN {X 0,Y 292.136,Z 630.258,A -85,B 0,C 180,E1 -17035.085,E2 -17035.085} C_VEL
LIN {X 0,Y 294.318,Z 616.265,A -85,B 0,C 180,E1 -17036.787,E2 -17036.787} C_VEL
LIN {X 0,Y 296.289,Z 602.681,A -85,B 0,C 180,E1 -17038.125,E2 -17038.125} C_VEL
LIN {X 0,Y 298.109,Z 588.017,A -85,B 0,C 180,E1 -17039.275,E2 -17039.275} C_VEL
LIN {X 0,Y 299.688,Z 572.899,A -85,B 0,C 180,E1 -17040.178,E2 -17040.178} C_VEL
LIN {X 0,Y 300.916,Z 556.68,A -85,B 0,C 180,E1 -17040.867,E2 -17040.867} C_VEL
LIN {X 0,Y 306.559,Z 446.079,A -85,B 0,C 180,E1 -17044.16,E2 -17044.16} C_VEL
LIN {X 0,Y 304.328,Z 432.908,A -85,B 0,C 180,E1 -17044.817,E2 -17044.817} C_VEL
LIN {X 0,Y 292.355,Z 403.525,A -85,B 0,C 180,E1 -17047.074,E2 -17047.074} C_VEL
LIN {X 0,Y 287.62,Z 392.468,A -85,B 0,C 180,E1 -17048.048,E2 -17048.048} C_VEL
LIN {X 0,Y 284.244,Z 379.704,A -85,B 0,C 180,E1 -17051.938,E2 -17051.938} C_VEL
LIN {X 0,Y 284.227,Z 379.707,A -85,B 0,C 180,E1 -17056.184,E2 -17056.184} C_VEL
LIN {X 0,Y 284.272,Z 379.702,A -85,B 0,C 180,E1 -17060.028,E2 -17060.028} C_VEL
LIN {X 0,Y 284.306,Z 379.696,A -85,B 0,C 180,E1 -17063.611,E2 -17063.611} C_VEL
LIN {X 0,Y 284.294,Z 379.696,A -85,B 0,C 180,E1 -17067.189,E2 -17067.189} C_VEL
LIN {X 0,Y 284.296,Z 379.697,A -85,B 0,C 180,E1 -17070.369,E2 -17070.369} C_VEL
LIN {X 0,Y 284.283,Z 379.696,A -85,B 0,C 180,E1 -17073.577,E2 -17073.577} C_VEL
LIN {X 0,Y 284.296,Z 379.696,A -85,B 0,C 180,E1 -17076.701,E2 -17076.701} C_VEL
LIN {X 0,Y 284.32,Z 379.693,A -85,B 0,C 180,E1 -17079.927,E2 -17079.927} C_VEL
LIN {X 0,Y 284.418,Z 379.681,A -85,B 0,C 180,E1 -17084.503,E2 -17084.503} C_VEL
LIN {X 0,Y 284.445,Z 379.671,A -85,B 0,C 180,E1 -17088.6,E2 -17088.6} C_VEL
LIN {X 0,Y 284.594,Z 379.654,A -85,B 0,C 180,E1 -17091.48,E2 -17091.48} C_VEL
LIN {X 0,Y 284.553,Z 379.665,A -85,B 0,C 180,E1 -17094.331,E2 -17094.331} C_VEL
LIN {X 0,Y 284.823,Z 379.629,A -85,B 0,C 180,E1 -17098.586,E2 -17098.586} C_VEL
LIN {X 0,Y 284.823,Z 379.63,A -85,B 0,C 180,E1 -17101.414,E2 -17101.414} C_VEL
LIN {X 0,Y 284.628,Z 379.653,A -85,B 0,C 180,E1 -17107.092,E2 -17107.092} C_VEL
LIN {X 0,Y 284.5,Z 379.67,A -85,B 0,C 180,E1 -17109.958,E2 -17109.958} C_VEL
LIN {X 0,Y 284.405,Z 379.683,A -85,B 0,C 180,E1 -17114.307,E2 -17114.307} C_VEL
LIN {X 0,Y 284.344,Z 379.686,A -85,B 0,C 180,E1 -17117.254,E2 -17117.254} C_VEL
LIN {X 0,Y 284.31,Z 379.695,A -85,B 0,C 180,E1 -17120.248,E2 -17120.248} C_VEL
LIN {X 0,Y 284.286,Z 379.699,A -85,B 0,C 180,E1 -17123.844,E2 -17123.844} C_VEL
LIN {X 0,Y 284.274,Z 379.695,A -85,B 0,C 180,E1 -17127.131,E2 -17127.131} C_VEL
LIN {X 0,Y 284.263,Z 379.701,A -85,B 0,C 180,E1 -17130.086,E2 -17130.086} C_VEL
LIN {X 0,Y 284.294,Z 379.692,A -85,B 0,C 180,E1 -17132.947,E2 -17132.947} C_VEL
LIN {X 0,Y 284.308,Z 379.693,A -85,B 0,C 180,E1 -17136.39,E2 -17136.39} C_VEL
LIN {X 0,Y 284.273,Z 379.699,A -85,B 0,C 180,E1 -17140.001,E2 -17140.001} C_VEL
LIN {X 0,Y 284.226,Z 379.704,A -85,B 0,C 180,E1 -17144.19,E2 -17144.19} C_VEL
LIN {X 0,Y 284.232,Z 379.703,A -85,B 0,C 180,E1 -17148.121,E2 -17148.121} C_VEL
LIN {X 0,Y 284.275,Z 379.697,A -85,B 0,C 180,E1 -17152.291,E2 -17152.291} C_VEL
LIN {X 0,Y 284.302,Z 379.695,A -85,B 0,C 180,E1 -17155.353,E2 -17155.353} C_VEL
LIN {X 0,Y 284.274,Z 379.694,A -85,B 0,C 180,E1 -17158.726,E2 -17158.726} C_VEL
LIN {X 0,Y 284.256,Z 379.702,A -85,B 0,C 180,E1 -17161.984,E2 -17161.984} C_VEL
LIN {X 0,Y 284.308,Z 379.694,A -85,B 0,C 180,E1 -17166.154,E2 -17166.154} C_VEL
LIN {X 0,Y 284.375,Z 379.688,A -85,B 0,C 180,E1 -17169.907,E2 -17169.907} C_VEL
LIN {X 0,Y 284.447,Z 379.665,A -85,B 0,C 180,E1 -17174.494,E2 -17174.494} C_VEL
LIN {X 0,Y 284.488,Z 379.67,A -85,B 0,C 180,E1 -17178.604,E2 -17178.604} C_VEL
LIN {X 0,Y 284.61,Z 379.659,A -85,B 0,C 180,E1 -17181.482,E2 -17181.482} C_VEL
LIN {X 0,Y 284.569,Z 379.654,A -85,B 0,C 180,E1 -17184.333,E2 -17184.333} C_VEL
LIN {X 0,Y 284.847,Z 379.626,A -85,B 0,C 180,E1 -17188.588,E2 -17188.588} C_VEL
LIN {X 0,Y 284.841,Z 379.629,A -85,B 0,C 180,E1 -17191.416,E2 -17191.416} C_VEL
LIN {X 0,Y 284.652,Z 379.653,A -85,B 0,C 180,E1 -17197.093,E2 -17197.093} C_VEL
LIN {X 0,Y 284.519,Z 379.669,A -85,B 0,C 180,E1 -17199.959,E2 -17199.959} C_VEL
LIN {X 0,Y 284.424,Z 379.677,A -85,B 0,C 180,E1 -17204.308,E2 -17204.308} C_VEL
LIN {X 0,Y 284.337,Z 379.688,A -85,B 0,C 180,E1 -17208.745,E2 -17208.745} C_VEL
LIN {X 0,Y 284.322,Z 379.693,A -85,B 0,C 180,E1 -17211.766,E2 -17211.766} C_VEL
LIN {X 0,Y 284.303,Z 379.694,A -85,B 0,C 180,E1 -17214.852,E2 -17214.852} C_VEL
LIN {X 0,Y 284.288,Z 379.698,A -85,B 0,C 180,E1 -17218.017,E2 -17218.017} C_VEL
LIN {X 0,Y 284.292,Z 379.699,A -85,B 0,C 180,E1 -17221.277,E2 -17221.277} C_VEL
LIN {X 0,Y 284.335,Z 379.759,A -85,B 0,C 180,E1 -17222.847,E2 -17222.847} C_VEL
LIN {X 0,Y 285.367,Z 382.531,A -85,B 0,C 180,E1 -17223.071,E2 -17223.071} C_VEL
LIN {X 0,Y 293.477,Z 398.692,A -85,B 0,C 180,E1 -17224.561,E2 -17224.561} C_VEL
LIN {X 0,Y 303.399,Z 422.056,A -85,B 0,C 180,E1 -17226.401,E2 -17226.401} C_VEL
LIN {X 0,Y 306.726,Z 430.366,A -85,B 0,C 180,E1 -17226.996,E2 -17226.996} C_VEL
LIN {X 0,Y 300.852,Z 543.699,A -85,B 0,C 180,E1 -17230.378,E2 -17230.378} C_VEL
LIN {X 0,Y 299.564,Z 559.648,A -85,B 0,C 180,E1 -17231.122,E2 -17231.122} C_VEL
LIN {X 0,Y 298.028,Z 575.454,A -85,B 0,C 180,E1 -17232.153,E2 -17232.153} C_VEL
LIN {X 0,Y 296.258,Z 589.724,A -85,B 0,C 180,E1 -17233.351,E2 -17233.351} C_VEL
LIN {X 0,Y 294.155,Z 604.761,A -85,B 0,C 180,E1 -17234.943,E2 -17234.943} C_VEL
LIN {X 0,Y 292.078,Z 618.199,A -85,B 0,C 180,E1 -17236.703,E2 -17236.703} C_VEL
LIN {X 0,Y 290.062,Z 630.642,A -85,B 0,C 180,E1 -17238.689,E2 -17238.689} C_VEL
LIN {X 0,Y 288.111,Z 642.021,A -85,B 0,C 180,E1 -17240.881,E2 -17240.881} C_VEL
LIN {X 0,Y 286.548,Z 651.444,A -85,B 0,C 180,E1 -17243.065,E2 -17243.065} C_VEL
LIN {X 0,Y 285.132,Z 660.096,A -85,B 0,C 180,E1 -17245.464,E2 -17245.464} C_VEL
LIN {X 0,Y 284.072,Z 667.429,A -85,B 0,C 180,E1 -17247.923,E2 -17247.923} C_VEL
LIN {X 0,Y 283.35,Z 673.199,A -85,B 0,C 180,E1 -17250.259,E2 -17250.259} C_VEL
LIN {X 0,Y 282.771,Z 678.414,A -85,B 0,C 180,E1 -17252.919,E2 -17252.919} C_VEL
LIN {X 0,Y 282.389,Z 681.601,A -85,B 0,C 180,E1 -17254.97,E2 -17254.97} C_VEL
LIN {X 0,Y 282.097,Z 685.076,A -85,B 0,C 180,E1 -17258.055,E2 -17258.055} C_VEL
LIN {X 0,Y 282.033,Z 685.74,A -85,B 0,C 180,E1 -17258.926,E2 -17258.926} C_VEL
LIN {X 0,Y 281.333,Z 686.587,A -85,B 0,C 180,E1 -17260.106,E2 -17260.106} C_VEL
LIN {X 0,Y 278.459,Z 687.549,A -85,B 0,C 180,E1 -17262.039,E2 -17262.039} C_VEL
LIN {X 0,Y 276.107,Z 687.901,A -85,B 0,C 180,E1 -17263.616,E2 -17263.616} C_VEL
LIN {X 0,Y 275.193,Z 687.877,A -85,B 0,C 180,E1 -17264.838,E2 -17264.838} C_VEL
LIN {X 0,Y 275.169,Z 687.807,A -85,B 0,C 180,E1 -17265.25,E2 -17265.25} C_VEL
LIN {X 0,Y 275.679,Z 686.754,A -85,B 0,C 180,E1 -17268.232,E2 -17268.232} C_VEL
LIN {X 0,Y 276.614,Z 684.432,A -85,B 0,C 180,E1 -17271.231,E2 -17271.231} C_VEL
LIN {X 0,Y 277.886,Z 680.849,A -85,B 0,C 180,E1 -17274.193,E2 -17274.193} C_VEL
LIN {X 0,Y 279.714,Z 675.959,A -85,B 0,C 180,E1 -17277.119,E2 -17277.119} C_VEL
LIN {X 0,Y 282.097,Z 669.671,A -85,B 0,C 180,E1 -17280,E2 -17280} C_VEL
LIN {X 0,Y 285.033,Z 661.786,A -85,B 0,C 180,E1 -17282.826,E2 -17282.826} C_VEL
LIN {X 0,Y 288.171,Z 653.469,A -85,B 0,C 180,E1 -17285.247,E2 -17285.247} C_VEL
LIN {X 0,Y 291.924,Z 643.108,A -85,B 0,C 180,E1 -17287.692,E2 -17287.692} C_VEL
LIN {X 0,Y 295.877,Z 631.539,A -85,B 0,C 180,E1 -17289.916,E2 -17289.916} C_VEL
LIN {X 0,Y 299.776,Z 619.301,A -85,B 0,C 180,E1 -17291.837,E2 -17291.837} C_VEL
LIN {X 0,Y 303.667,Z 605.665,A -85,B 0,C 180,E1 -17293.576,E2 -17293.576} C_VEL
LIN {X 0,Y 307.407,Z 591.14,A -85,B 0,C 180,E1 -17295.073,E2 -17295.073} C_VEL
LIN {X 0,Y 310.204,Z 578.473,A -85,B 0,C 180,E1 -17296.113,E2 -17296.113} C_VEL
LIN {X 0,Y 312.914,Z 563.946,A -85,B 0,C 180,E1 -17297.06,E2 -17297.06} C_VEL
LIN {X 0,Y 315.473,Z 546.988,A -85,B 0,C 180,E1 -17297.879,E2 -17297.879} C_VEL
LIN {X 0,Y 326.511,Z 449.808,A -85,B 0,C 180,E1 -17301.117,E2 -17301.117} C_VEL
LIN {X 0,Y 323.592,Z 443.354,A -85,B 0,C 180,E1 -17302.524,E2 -17302.524} C_VEL
LIN {X 0,Y 320.416,Z 437.171,A -85,B 0,C 180,E1 -17304.23,E2 -17304.23} C_VEL
LIN {X 0,Y 317.491,Z 432.188,A -85,B 0,C 180,E1 -17306.051,E2 -17306.051} C_VEL
LIN {X 0,Y 314.958,Z 428.084,A -85,B 0,C 180,E1 -17308.009,E2 -17308.009} C_VEL
LIN {X 0,Y 312.551,Z 424.536,A -85,B 0,C 180,E1 -17310.588,E2 -17310.588} C_VEL
LIN {X 0,Y 311.064,Z 422.773,A -85,B 0,C 180,E1 -17313.282,E2 -17313.282} C_VEL
LIN {X 0,Y 310.762,Z 422.823,A -85,B 0,C 180,E1 -17316.015,E2 -17316.015} C_VEL
LIN {X 0,Y 311.398,Z 424.557,A -85,B 0,C 180,E1 -17318.472,E2 -17318.472} C_VEL
LIN {X 0,Y 313.233,Z 427.56,A -85,B 0,C 180,E1 -17321.138,E2 -17321.138} C_VEL
LIN {X 0,Y 316.324,Z 433.614,A -85,B 0,C 180,E1 -17323.964,E2 -17323.964} C_VEL
LIN {X 0,Y 318.77,Z 438.667,A -85,B 0,C 180,E1 -17325.677,E2 -17325.677} C_VEL
LIN {X 0,Y 321.311,Z 444.268,A -85,B 0,C 180,E1 -17327.21,E2 -17327.21} C_VEL
LIN {X 0,Y 324.082,Z 451.194,A -85,B 0,C 180,E1 -17328.722,E2 -17328.722} C_VEL
LIN {X 0,Y 326.087,Z 456.65,A -85,B 0,C 180,E1 -17329.714,E2 -17329.714} C_VEL
LIN {X 0,Y 314.684,Z 557.566,A -85,B 0,C 180,E1 -17333.063,E2 -17333.063} C_VEL
LIN {X 0,Y 312.038,Z 574.485,A -85,B 0,C 180,E1 -17333.854,E2 -17333.854} C_VEL
LIN {X 0,Y 309.033,Z 589.152,A -85,B 0,C 180,E1 -17334.753,E2 -17334.753} C_VEL
LIN {X 0,Y 305.681,Z 603.386,A -85,B 0,C 180,E1 -17335.894,E2 -17335.894} C_VEL
LIN {X 0,Y 302.178,Z 616.557,A -85,B 0,C 180,E1 -17337.209,E2 -17337.209} C_VEL
LIN {X 0,Y 298.425,Z 629.515,A -85,B 0,C 180,E1 -17338.793,E2 -17338.793} C_VEL
LIN {X 0,Y 294.375,Z 642.224,A -85,B 0,C 180,E1 -17340.695,E2 -17340.695} C_VEL
LIN {X 0,Y 290.227,Z 654.682,A -85,B 0,C 180,E1 -17342.995,E2 -17342.995} C_VEL
LIN {X 0,Y 286.634,Z 665.127,A -85,B 0,C 180,E1 -17345.364,E2 -17345.364} C_VEL
LIN {X 0,Y 283.212,Z 675.067,A -85,B 0,C 180,E1 -17348.145,E2 -17348.145} C_VEL
LIN {X 0,Y 281.094,Z 681.365,A -85,B 0,C 180,E1 -17350.271,E2 -17350.271} C_VEL
LIN {X 0,Y 278.628,Z 688.483,A -85,B 0,C 180,E1 -17353.211,E2 -17353.211} C_VEL
LIN {X 0,Y 277.133,Z 693.873,A -85,B 0,C 180,E1 -17356.057,E2 -17356.057} C_VEL
LIN {X 0,Y 276.206,Z 697.112,A -85,B 0,C 180,E1 -17358.253,E2 -17358.253} C_VEL
LIN {X 0,Y 275.554,Z 700.365,A -85,B 0,C 180,E1 -17361.195,E2 -17361.195} C_VEL
LIN {X 0,Y 275.235,Z 702.399,A -85,B 0,C 180,E1 -17364.136,E2 -17364.136} C_VEL
LIN {X 0,Y 275.233,Z 703.208,A -85,B 0,C 180,E1 -17367.071,E2 -17367.071} C_VEL
LIN {X 0,Y 275.279,Z 702.738,A -85,B 0,C 180,E1 -17369.998,E2 -17369.998} C_VEL
LIN {X 0,Y 275.328,Z 701.007,A -85,B 0,C 180,E1 -17372.924,E2 -17372.924} C_VEL
LIN {X 0,Y 275.33,Z 697.957,A -85,B 0,C 180,E1 -17375.858,E2 -17375.858} C_VEL
LIN {X 0,Y 275.544,Z 693.51,A -85,B 0,C 180,E1 -17378.801,E2 -17378.801} C_VEL
LIN {X 0,Y 276,Z 687.521,A -85,B 0,C 180,E1 -17381.752,E2 -17381.752} C_VEL
LIN {X 0,Y 276.852,Z 680.923,A -85,B 0,C 180,E1 -17384.328,E2 -17384.328} C_VEL
LIN {X 0,Y 278.029,Z 672.873,A -85,B 0,C 180,E1 -17386.897,E2 -17386.897} C_VEL
LIN {X 0,Y 279.605,Z 663.123,A -85,B 0,C 180,E1 -17389.451,E2 -17389.451} C_VEL
LIN {X 0,Y 281.371,Z 653.17,A -85,B 0,C 180,E1 -17391.616,E2 -17391.616} C_VEL
LIN {X 0,Y 283.353,Z 641.3,A -85,B 0,C 180,E1 -17393.766,E2 -17393.766} C_VEL
LIN {X 0,Y 285.39,Z 629.602,A -85,B 0,C 180,E1 -17395.525,E2 -17395.525} C_VEL
LIN {X 0,Y 287.624,Z 615.504,A -85,B 0,C 180,E1 -17397.265,E2 -17397.265} C_VEL
LIN {X 0,Y 289.68,Z 601.805,A -85,B 0,C 180,E1 -17398.628,E2 -17398.628} C_VEL
LIN {X 0,Y 291.543,Z 587.07,A -85,B 0,C 180,E1 -17399.794,E2 -17399.794} C_VEL
LIN {X 0,Y 293.15,Z 571.572,A -85,B 0,C 180,E1 -17400.724,E2 -17400.724} C_VEL
LIN {X 0,Y 294.425,Z 554.907,A -85,B 0,C 180,E1 -17401.424,E2 -17401.424} C_VEL
LIN {X 0,Y 300.082,Z 446.897,A -85,B 0,C 180,E1 -17404.719,E2 -17404.719} C_VEL
LIN {X 0,Y 298.192,Z 435.448,A -85,B 0,C 180,E1 -17405.308,E2 -17405.308} C_VEL
LIN {X 0,Y 286.549,Z 406.752,A -85,B 0,C 180,E1 -17407.573,E2 -17407.573} C_VEL
LIN {X 0,Y 280.321,Z 392.32,A -85,B 0,C 180,E1 -17408.866,E2 -17408.866} C_VEL
LIN {X 0,Y 277.165,Z 380.586,A -85,B 0,C 180,E1 -17412.545,E2 -17412.545} C_VEL
LIN {X 0,Y 277.181,Z 380.583,A -85,B 0,C 180,E1 -17416.797,E2 -17416.797} C_VEL
LIN {X 0,Y 277.204,Z 380.581,A -85,B 0,C 180,E1 -17420.667,E2 -17420.667} C_VEL
LIN {X 0,Y 277.265,Z 380.575,A -85,B 0,C 180,E1 -17424.339,E2 -17424.339} C_VEL
LIN {X 0,Y 277.225,Z 380.579,A -85,B 0,C 180,E1 -17427.834,E2 -17427.834} C_VEL
LIN {X 0,Y 277.203,Z 380.578,A -85,B 0,C 180,E1 -17431.203,E2 -17431.203} C_VEL
LIN {X 0,Y 277.221,Z 380.575,A -85,B 0,C 180,E1 -17434.471,E2 -17434.471} C_VEL
LIN {X 0,Y 277.235,Z 380.576,A -85,B 0,C 180,E1 -17437.651,E2 -17437.651} C_VEL
LIN {X 0,Y 277.268,Z 380.564,A -85,B 0,C 180,E1 -17440.761,E2 -17440.761} C_VEL
LIN {X 0,Y 277.363,Z 380.559,A -85,B 0,C 180,E1 -17445.322,E2 -17445.322} C_VEL
LIN {X 0,Y 277.44,Z 380.543,A -85,B 0,C 180,E1 -17449.787,E2 -17449.787} C_VEL
LIN {X 0,Y 277.586,Z 380.53,A -85,B 0,C 180,E1 -17452.728,E2 -17452.728} C_VEL
LIN {X 0,Y 277.79,Z 380.506,A -85,B 0,C 180,E1 -17458.551,E2 -17458.551} C_VEL
LIN {X 0,Y 277.79,Z 380.506,A -85,B 0,C 180,E1 -17461.45,E2 -17461.45} C_VEL
LIN {X 0,Y 277.587,Z 380.531,A -85,B 0,C 180,E1 -17467.273,E2 -17467.273} C_VEL
LIN {X 0,Y 277.44,Z 380.549,A -85,B 0,C 180,E1 -17470.214,E2 -17470.214} C_VEL
LIN {X 0,Y 277.363,Z 380.558,A -85,B 0,C 180,E1 -17474.678,E2 -17474.678} C_VEL
LIN {X 0,Y 277.269,Z 380.568,A -85,B 0,C 180,E1 -17479.24,E2 -17479.24} C_VEL
LIN {X 0,Y 277.248,Z 380.574,A -85,B 0,C 180,E1 -17483.928,E2 -17483.928} C_VEL
LIN {X 0,Y 277.224,Z 380.574,A -85,B 0,C 180,E1 -17487.471,E2 -17487.471} C_VEL
LIN {X 0,Y 277.217,Z 380.577,A -85,B 0,C 180,E1 -17490.467,E2 -17490.467} C_VEL
LIN {X 0,Y 277.236,Z 380.573,A -85,B 0,C 180,E1 -17493.898,E2 -17493.898} C_VEL
LIN {X 0,Y 277.241,Z 380.574,A -85,B 0,C 180,E1 -17497.474,E2 -17497.474} C_VEL
LIN {X 0,Y 277.175,Z 380.58,A -85,B 0,C 180,E1 -17501.243,E2 -17501.243} C_VEL
LIN {X 0,Y 277.166,Z 380.582,A -85,B 0,C 180,E1 -17505.234,E2 -17505.234} C_VEL
LIN {X 0,Y 277.17,Z 380.581,A -85,B 0,C 180,E1 -17508.76,E2 -17508.76} C_VEL
LIN {X 0,Y 277.226,Z 380.574,A -85,B 0,C 180,E1 -17512.527,E2 -17512.527} C_VEL
LIN {X 0,Y 277.241,Z 380.574,A -85,B 0,C 180,E1 -17516.106,E2 -17516.106} C_VEL
LIN {X 0,Y 277.224,Z 380.575,A -85,B 0,C 180,E1 -17519.537,E2 -17519.537} C_VEL
LIN {X 0,Y 277.247,Z 380.572,A -85,B 0,C 180,E1 -17522.855,E2 -17522.855} C_VEL
LIN {X 0,Y 277.269,Z 380.571,A -85,B 0,C 180,E1 -17526.077,E2 -17526.077} C_VEL
LIN {X 0,Y 277.323,Z 380.562,A -85,B 0,C 180,E1 -17530.767,E2 -17530.767} C_VEL
LIN {X 0,Y 277.41,Z 380.542,A -85,B 0,C 180,E1 -17535.327,E2 -17535.327} C_VEL
LIN {X 0,Y 277.461,Z 380.55,A -85,B 0,C 180,E1 -17539.789,E2 -17539.789} C_VEL
LIN {X 0,Y 277.602,Z 380.526,A -85,B 0,C 180,E1 -17542.73,E2 -17542.73} C_VEL
LIN {X 0,Y 277.813,Z 380.503,A -85,B 0,C 180,E1 -17548.553,E2 -17548.553} C_VEL
LIN {X 0,Y 277.808,Z 380.505,A -85,B 0,C 180,E1 -17551.452,E2 -17551.452} C_VEL
LIN {X 0,Y 277.61,Z 380.531,A -85,B 0,C 180,E1 -17557.274,E2 -17557.274} C_VEL
LIN {X 0,Y 277.462,Z 380.546,A -85,B 0,C 180,E1 -17560.215,E2 -17560.215} C_VEL
LIN {X 0,Y 277.376,Z 380.554,A -85,B 0,C 180,E1 -17564.679,E2 -17564.679} C_VEL
LIN {X 0,Y 277.305,Z 380.566,A -85,B 0,C 180,E1 -17569.239,E2 -17569.239} C_VEL
LIN {X 0,Y 277.283,Z 380.57,A -85,B 0,C 180,E1 -17573.927,E2 -17573.927} C_VEL
LIN {X 0,Y 277.274,Z 380.572,A -85,B 0,C 180,E1 -17577.483,E2 -17577.483} C_VEL
LIN {X 0,Y 277.237,Z 380.579,A -85,B 0,C 180,E1 -17581.738,E2 -17581.738} C_VEL
LIN {X 0,Y 277.24,Z 380.578,A -85,B 0,C 180,E1 -17582.059,E2 -17582.059} C_VEL
LIN {X 0,Y 278.363,Z 383.598,A -85,B 0,C 180,E1 -17582.316,E2 -17582.316} C_VEL
LIN {X 0,Y 287.79,Z 402.182,A -85,B 0,C 180,E1 -17584.094,E2 -17584.094} C_VEL
LIN {X 0,Y 297.565,Z 425.385,A -85,B 0,C 180,E1 -17585.956,E2 -17585.956} C_VEL
LIN {X 0,Y 300.317,Z 432.395,A -85,B 0,C 180,E1 -17586.469,E2 -17586.469} C_VEL
LIN {X 0,Y 294.279,Z 543.554,A -85,B 0,C 180,E1 -17589.862,E2 -17589.862} C_VEL
LIN {X 0,Y 293.028,Z 559.199,A -85,B 0,C 180,E1 -17590.602,E2 -17590.602} C_VEL
LIN {X 0,Y 291.457,Z 574.779,A -85,B 0,C 180,E1 -17591.624,E2 -17591.624} C_VEL
LIN {X 0,Y 289.596,Z 589.596,A -85,B 0,C 180,E1 -17592.885,E2 -17592.885} C_VEL
LIN {X 0,Y 287.578,Z 603.54,A -85,B 0,C 180,E1 -17594.37,E2 -17594.37} C_VEL
LIN {X 0,Y 285.395,Z 617.445,A -85,B 0,C 180,E1 -17596.201,E2 -17596.201} C_VEL
LIN {X 0,Y 283.359,Z 629.697,A -85,B 0,C 180,E1 -17598.168,E2 -17598.168} C_VEL
LIN {X 0,Y 281.393,Z 640.66,A -85,B 0,C 180,E1 -17600.28,E2 -17600.28} C_VEL
LIN {X 0,Y 279.791,Z 650.185,A -85,B 0,C 180,E1 -17602.473,E2 -17602.473} C_VEL
LIN {X 0,Y 278.301,Z 659.115,A -85,B 0,C 180,E1 -17604.934,E2 -17604.934} C_VEL
LIN {X 0,Y 277.216,Z 666.151,A -85,B 0,C 180,E1 -17607.254,E2 -17607.254} C_VEL
LIN {X 0,Y 276.386,Z 672.562,A -85,B 0,C 180,E1 -17609.835,E2 -17609.835} C_VEL
LIN {X 0,Y 275.736,Z 678.204,A -85,B 0,C 180,E1 -17612.691,E2 -17612.691} C_VEL
LIN {X 0,Y 275.267,Z 681.853,A -85,B 0,C 180,E1 -17615.085,E2 -17615.085} C_VEL
LIN {X 0,Y 275.039,Z 684.63,A -85,B 0,C 180,E1 -17617.462,E2 -17617.462} C_VEL
LIN {X 0,Y 274.921,Z 686.957,A -85,B 0,C 180,E1 -17620.589,E2 -17620.589} C_VEL
LIN {X 0,Y 275.022,Z 687.868,A -85,B 0,C 180,E1 -17623.674,E2 -17623.674} C_VEL
LIN {X 0,Y 275.169,Z 687.807,A -85,B 0,C 180,E1 -17625.25,E2 -17625.25} C_VEL
LIN {X 0,Y 274.698,Z 687.555,A -85,B 0,C 180,E1 -17626.475,E2 -17626.475} C_VEL
LIN {X 0,Y 272.229,Z 686.861,A -85,B 0,C 180,E1 -17628.484,E2 -17628.484} C_VEL
LIN {X 0,Y 270.247,Z 685.989,A -85,B 0,C 180,E1 -17630.106,E2 -17630.106} C_VEL
LIN {X 0,Y 269.645,Z 685.074,A -85,B 0,C 180,E1 -17631.344,E2 -17631.344} C_VEL
LIN {X 0,Y 269.731,Z 684.684,A -85,B 0,C 180,E1 -17631.757,E2 -17631.757} C_VEL
LIN {X 0,Y 271.131,Z 681.139,A -85,B 0,C 180,E1 -17634.794,E2 -17634.794} C_VEL
LIN {X 0,Y 273.126,Z 676.279,A -85,B 0,C 180,E1 -17637.788,E2 -17637.788} C_VEL
LIN {X 0,Y 275.685,Z 670.006,A -85,B 0,C 180,E1 -17640.73,E2 -17640.73} C_VEL
LIN {X 0,Y 278.88,Z 662.214,A -85,B 0,C 180,E1 -17643.612,E2 -17643.612} C_VEL
LIN {X 0,Y 282.351,Z 653.536,A -85,B 0,C 180,E1 -17646.171,E2 -17646.171} C_VEL
LIN {X 0,Y 286.05,Z 644.025,A -85,B 0,C 180,E1 -17648.477,E2 -17648.477} C_VEL
LIN {X 0,Y 289.747,Z 634.021,A -85,B 0,C 180,E1 -17650.481,E2 -17650.481} C_VEL
LIN {X 0,Y 293.811,Z 622.171,A -85,B 0,C 180,E1 -17652.432,E2 -17652.432} C_VEL
LIN {X 0,Y 297.585,Z 610.139,A -85,B 0,C 180,E1 -17654.086,E2 -17654.086} C_VEL
LIN {X 0,Y 301.318,Z 596.918,A -85,B 0,C 180,E1 -17655.559,E2 -17655.559} C_VEL
LIN {X 0,Y 304.993,Z 581.772,A -85,B 0,C 180,E1 -17656.913,E2 -17656.913} C_VEL
LIN {X 0,Y 308.062,Z 567.043,A -85,B 0,C 180,E1 -17657.937,E2 -17657.937} C_VEL
LIN {X 0,Y 310.699,Z 551.426,A -85,B 0,C 180,E1 -17658.744,E2 -17658.744} C_VEL
LIN {X 0,Y 313.114,Z 531.817,A -85,B 0,C 180,E1 -17659.46,E2 -17659.46} C_VEL
LIN {X 0,Y 322.574,Z 453.264,A -85,B 0,C 180,E1 -17662.103,E2 -17662.103} C_VEL
LIN {X 0,Y 319.746,Z 446.993,A -85,B 0,C 180,E1 -17663.627,E2 -17663.627} C_VEL
LIN {X 0,Y 316.898,Z 441.341,A -85,B 0,C 180,E1 -17665.37,E2 -17665.37} C_VEL
LIN {X 0,Y 315.11,Z 438.195,A -85,B 0,C 180,E1 -17666.625,E2 -17666.625} C_VEL
LIN {X 0,Y 313.078,Z 434.696,A -85,B 0,C 180,E1 -17668.327,E2 -17668.327} C_VEL
LIN {X 0,Y 311.005,Z 431.446,A -85,B 0,C 180,E1 -17670.661,E2 -17670.661} C_VEL
LIN {X 0,Y 309.545,Z 429.699,A -85,B 0,C 180,E1 -17673.393,E2 -17673.393} C_VEL
LIN {X 0,Y 309.257,Z 429.67,A -85,B 0,C 180,E1 -17675.674,E2 -17675.674} C_VEL
LIN {X 0,Y 309.767,Z 431.208,A -85,B 0,C 180,E1 -17678.108,E2 -17678.108} C_VEL
LIN {X 0,Y 311.48,Z 434.286,A -85,B 0,C 180,E1 -17680.869,E2 -17680.869} C_VEL
LIN {X 0,Y 314.102,Z 439.799,A -85,B 0,C 180,E1 -17683.482,E2 -17683.482} C_VEL
LIN {X 0,Y 316.309,Z 444.746,A -85,B 0,C 180,E1 -17685.183,E2 -17685.183} C_VEL
LIN {X 0,Y 318.678,Z 450.372,A -85,B 0,C 180,E1 -17686.742,E2 -17686.742} C_VEL
LIN {X 0,Y 321.418,Z 457.611,A -85,B 0,C 180,E1 -17688.318,E2 -17688.318} C_VEL
LIN {X 0,Y 322.117,Z 459.987,A -85,B 0,C 180,E1 -17688.734,E2 -17688.734} C_VEL
LIN {X 0,Y 310.469,Z 557.578,A -85,B 0,C 180,E1 -17692.015,E2 -17692.015} C_VEL
LIN {X 0,Y 307.557,Z 574.772,A -85,B 0,C 180,E1 -17692.832,E2 -17692.832} C_VEL
LIN {X 0,Y 303.954,Z 591.061,A -85,B 0,C 180,E1 -17693.869,E2 -17693.869} C_VEL
LIN {X 0,Y 300.53,Z 604.698,A -85,B 0,C 180,E1 -17695.002,E2 -17695.002} C_VEL
LIN {X 0,Y 296.527,Z 618.813,A -85,B 0,C 180,E1 -17696.472,E2 -17696.472} C_VEL
LIN {X 0,Y 292.913,Z 630.271,A -85,B 0,C 180,E1 -17697.935,E2 -17697.935} C_VEL
LIN {X 0,Y 289.01,Z 641.849,A -85,B 0,C 180,E1 -17699.694,E2 -17699.694} C_VEL
LIN {X 0,Y 285.206,Z 652.645,A -85,B 0,C 180,E1 -17701.681,E2 -17701.681} C_VEL
LIN {X 0,Y 281.29,Z 663.35,A -85,B 0,C 180,E1 -17704.086,E2 -17704.086} C_VEL
LIN {X 0,Y 277.941,Z 672.356,A -85,B 0,C 180,E1 -17706.529,E2 -17706.529} C_VEL
LIN {X 0,Y 275.151,Z 679.944,A -85,B 0,C 180,E1 -17709.046,E2 -17709.046} C_VEL
LIN {X 0,Y 272.495,Z 687.132,A -85,B 0,C 180,E1 -17711.969,E2 -17711.969} C_VEL
LIN {X 0,Y 270.872,Z 691.536,A -85,B 0,C 180,E1 -17714.189,E2 -17714.189} C_VEL
LIN {X 0,Y 269.534,Z 696.25,A -85,B 0,C 180,E1 -17717.193,E2 -17717.193} C_VEL
LIN {X 0,Y 268.787,Z 698.939,A -85,B 0,C 180,E1 -17719.452,E2 -17719.452} C_VEL
LIN {X 0,Y 268.253,Z 701.457,A -85,B 0,C 180,E1 -17722.471,E2 -17722.471} C_VEL
LIN {X 0,Y 268.103,Z 702.772,A -85,B 0,C 180,E1 -17725.487,E2 -17725.487} C_VEL
LIN {X 0,Y 268.184,Z 702.874,A -85,B 0,C 180,E1 -17728.496,E2 -17728.496} C_VEL
LIN {X 0,Y 268.207,Z 701.675,A -85,B 0,C 180,E1 -17731.499,E2 -17731.499} C_VEL
LIN {X 0,Y 268.235,Z 700.591,A -85,B 0,C 180,E1 -17733.002,E2 -17733.002} C_VEL
LIN {X 0,Y 268.24,Z 697.418,A -85,B 0,C 180,E1 -17736.013,E2 -17736.013} C_VEL
LIN {X 0,Y 268.462,Z 692.837,A -85,B 0,C 180,E1 -17739.035,E2 -17739.035} C_VEL
LIN {X 0,Y 268.996,Z 686.718,A -85,B 0,C 180,E1 -17742.062,E2 -17742.062} C_VEL
LIN {X 0,Y 269.856,Z 679.97,A -85,B 0,C 180,E1 -17744.707,E2 -17744.707} C_VEL
LIN {X 0,Y 271.13,Z 671.764,A -85,B 0,C 180,E1 -17747.341,E2 -17747.341} C_VEL
LIN {X 0,Y 272.824,Z 661.838,A -85,B 0,C 180,E1 -17749.955,E2 -17749.955} C_VEL
LIN {X 0,Y 274.688,Z 651.683,A -85,B 0,C 180,E1 -17752.169,E2 -17752.169} C_VEL
LIN {X 0,Y 276.556,Z 640.667,A -85,B 0,C 180,E1 -17754.188,E2 -17754.188} C_VEL
LIN {X 0,Y 278.657,Z 628.896,A -85,B 0,C 180,E1 -17755.987,E2 -17755.987} C_VEL
LIN {X 0,Y 280.714,Z 616.297,A -85,B 0,C 180,E1 -17757.589,E2 -17757.589} C_VEL
LIN {X 0,Y 282.783,Z 602.845,A -85,B 0,C 180,E1 -17758.986,E2 -17758.986} C_VEL
LIN {X 0,Y 284.703,Z 588.255,A -85,B 0,C 180,E1 -17760.194,E2 -17760.194} C_VEL
LIN {X 0,Y 286.419,Z 572.748,A -85,B 0,C 180,E1 -17761.168,E2 -17761.168} C_VEL
LIN {X 0,Y 287.746,Z 556.82,A -85,B 0,C 180,E1 -17761.879,E2 -17761.879} C_VEL
LIN {X 0,Y 293.712,Z 448.076,A -85,B 0,C 180,E1 -17765.285,E2 -17765.285} C_VEL
LIN {X 0,Y 292.017,Z 437.828,A -85,B 0,C 180,E1 -17765.831,E2 -17765.831} C_VEL
LIN {X 0,Y 280.651,Z 409.817,A -85,B 0,C 180,E1 -17768.089,E2 -17768.089} C_VEL
LIN {X 0,Y 272.945,Z 392.169,A -85,B 0,C 180,E1 -17769.725,E2 -17769.725} C_VEL
LIN {X 0,Y 270.142,Z 381.46,A -85,B 0,C 180,E1 -17773.175,E2 -17773.175} C_VEL
LIN {X 0,Y 270.14,Z 381.46,A -85,B 0,C 180,E1 -17777.436,E2 -17777.436} C_VEL
LIN {X 0,Y 270.181,Z 381.455,A -85,B 0,C 180,E1 -17781.37,E2 -17781.37} C_VEL
LIN {X 0,Y 270.185,Z 381.454,A -85,B 0,C 180,E1 -17785.093,E2 -17785.093} C_VEL
LIN {X 0,Y 270.158,Z 381.456,A -85,B 0,C 180,E1 -17789.14,E2 -17789.14} C_VEL
LIN {X 0,Y 270.175,Z 381.457,A -85,B 0,C 180,E1 -17792.176,E2 -17792.176} C_VEL
LIN {X 0,Y 270.171,Z 381.453,A -85,B 0,C 180,E1 -17795.562,E2 -17795.562} C_VEL
LIN {X 0,Y 270.208,Z 381.446,A -85,B 0,C 180,E1 -17800.238,E2 -17800.238} C_VEL
LIN {X 0,Y 270.332,Z 381.435,A -85,B 0,C 180,E1 -17804.932,E2 -17804.932} C_VEL
LIN {X 0,Y 270.372,Z 381.422,A -85,B 0,C 180,E1 -17809.517,E2 -17809.517} C_VEL
LIN {X 0,Y 270.548,Z 381.408,A -85,B 0,C 180,E1 -17812.537,E2 -17812.537} C_VEL
LIN {X 0,Y 270.755,Z 381.382,A -85,B 0,C 180,E1 -17818.513,E2 -17818.513} C_VEL
LIN {X 0,Y 270.755,Z 381.382,A -85,B 0,C 180,E1 -17821.488,E2 -17821.488} C_VEL
LIN {X 0,Y 270.548,Z 381.408,A -85,B 0,C 180,E1 -17827.463,E2 -17827.463} C_VEL
LIN {X 0,Y 270.372,Z 381.427,A -85,B 0,C 180,E1 -17830.484,E2 -17830.484} C_VEL
LIN {X 0,Y 270.333,Z 381.433,A -85,B 0,C 180,E1 -17835.069,E2 -17835.069} C_VEL
LIN {X 0,Y 270.209,Z 381.45,A -85,B 0,C 180,E1 -17839.763,E2 -17839.763} C_VEL
LIN {X 0,Y 270.172,Z 381.451,A -85,B 0,C 180,E1 -17844.438,E2 -17844.438} C_VEL
LIN {X 0,Y 270.173,Z 381.456,A -85,B 0,C 180,E1 -17847.92,E2 -17847.92} C_VEL
LIN {X 0,Y 270.158,Z 381.456,A -85,B 0,C 180,E1 -17851.352,E2 -17851.352} C_VEL
LIN {X 0,Y 270.187,Z 381.448,A -85,B 0,C 180,E1 -17854.908,E2 -17854.908} C_VEL
LIN {X 0,Y 270.189,Z 381.451,A -85,B 0,C 180,E1 -17858.712,E2 -17858.712} C_VEL
LIN {X 0,Y 270.14,Z 381.454,A -85,B 0,C 180,E1 -17863.247,E2 -17863.247} C_VEL
LIN {X 0,Y 270.143,Z 381.459,A -85,B 0,C 180,E1 -17867.44,E2 -17867.44} C_VEL
LIN {X 0,Y 270.145,Z 381.454,A -85,B 0,C 180,E1 -17871.367,E2 -17871.367} C_VEL
LIN {X 0,Y 270.192,Z 381.452,A -85,B 0,C 180,E1 -17875.096,E2 -17875.096} C_VEL
LIN {X 0,Y 270.167,Z 381.451,A -85,B 0,C 180,E1 -17879.144,E2 -17879.144} C_VEL
LIN {X 0,Y 270.184,Z 381.454,A -85,B 0,C 180,E1 -17882.179,E2 -17882.179} C_VEL
LIN {X 0,Y 270.187,Z 381.453,A -85,B 0,C 180,E1 -17885.563,E2 -17885.563} C_VEL
LIN {X 0,Y 270.259,Z 381.443,A -85,B 0,C 180,E1 -17890.244,E2 -17890.244} C_VEL
LIN {X 0,Y 270.377,Z 381.415,A -85,B 0,C 180,E1 -17894.936,E2 -17894.936} C_VEL
LIN {X 0,Y 270.413,Z 381.426,A -85,B 0,C 180,E1 -17899.52,E2 -17899.52} C_VEL
LIN {X 0,Y 270.563,Z 381.403,A -85,B 0,C 180,E1 -17902.54,E2 -17902.54} C_VEL
LIN {X 0,Y 270.778,Z 381.379,A -85,B 0,C 180,E1 -17908.515,E2 -17908.515} C_VEL
LIN {X 0,Y 270.773,Z 381.381,A -85,B 0,C 180,E1 -17911.489,E2 -17911.489} C_VEL
LIN {X 0,Y 270.571,Z 381.409,A -85,B 0,C 180,E1 -17917.464,E2 -17917.464} C_VEL
LIN {X 0,Y 270.414,Z 381.423,A -85,B 0,C 180,E1 -17920.484,E2 -17920.484} C_VEL
LIN {X 0,Y 270.343,Z 381.431,A -85,B 0,C 180,E1 -17925.07,E2 -17925.07} C_VEL
LIN {X 0,Y 270.255,Z 381.448,A -85,B 0,C 180,E1 -17929.761,E2 -17929.761} C_VEL
LIN {X 0,Y 270.206,Z 381.45,A -85,B 0,C 180,E1 -17934.594,E2 -17934.594} C_VEL
LIN {X 0,Y 270.203,Z 381.453,A -85,B 0,C 180,E1 -17937.918,E2 -17937.918} C_VEL
LIN {X 0,Y 270.249,Z 381.577,A -85,B 0,C 180,E1 -17941.257,E2 -17941.257} C_VEL
LIN {X 0,Y 271.215,Z 384.283,A -85,B 0,C 180,E1 -17941.489,E2 -17941.489} C_VEL
LIN {X 0,Y 281.295,Z 403.934,A -85,B 0,C 180,E1 -17943.461,E2 -17943.461} C_VEL
LIN {X 0,Y 291.235,Z 427.378,A -85,B 0,C 180,E1 -17945.394,E2 -17945.394} C_VEL
LIN {X 0,Y 293.778,Z 433.687,A -85,B 0,C 180,E1 -17945.882,E2 -17945.882} C_VEL
LIN {X 0,Y 287.689,Z 544.022,A -85,B 0,C 180,E1 -17949.351,E2 -17949.351} C_VEL
LIN {X 0,Y 286.33,Z 559.94,A -85,B 0,C 180,E1 -17950.13,E2 -17950.13} C_VEL
LIN {X 0,Y 284.755,Z 575.247,A -85,B 0,C 180,E1 -17951.169,E2 -17951.169} C_VEL
LIN {X 0,Y 282.843,Z 590.068,A -85,B 0,C 180,E1 -17952.466,E2 -17952.466} C_VEL
LIN {X 0,Y 280.729,Z 604.252,A -85,B 0,C 180,E1 -17954.023,E2 -17954.023} C_VEL
LIN {X 0,Y 278.562,Z 617.524,A -85,B 0,C 180,E1 -17955.815,E2 -17955.815} C_VEL
LIN {X 0,Y 276.344,Z 630.485,A -85,B 0,C 180,E1 -17957.954,E2 -17957.954} C_VEL
LIN {X 0,Y 274.263,Z 641.932,A -85,B 0,C 180,E1 -17960.244,E2 -17960.244} C_VEL
LIN {X 0,Y 272.571,Z 651.558,A -85,B 0,C 180,E1 -17962.565,E2 -17962.565} C_VEL
LIN {X 0,Y 271.014,Z 660.673,A -85,B 0,C 180,E1 -17965.214,E2 -17965.214} C_VEL
LIN {X 0,Y 269.925,Z 667.835,A -85,B 0,C 180,E1 -17967.74,E2 -17967.74} C_VEL
LIN {X 0,Y 269.163,Z 673.734,A -85,B 0,C 180,E1 -17970.257,E2 -17970.257} C_VEL
LIN {X 0,Y 268.596,Z 678.593,A -85,B 0,C 180,E1 -17972.831,E2 -17972.831} C_VEL
LIN {X 0,Y 268.17,Z 682.097,A -85,B 0,C 180,E1 -17975.208,E2 -17975.208} C_VEL
LIN {X 0,Y 267.986,Z 684.022,A -85,B 0,C 180,E1 -17976.835,E2 -17976.835} C_VEL
LIN {X 0,Y 267.813,Z 686.716,A -85,B 0,C 180,E1 -17980.053,E2 -17980.053} C_VEL
LIN {X 0,Y 267.885,Z 687.975,A -85,B 0,C 180,E1 -17983.226,E2 -17983.226} C_VEL
LIN {X 0,Y 268.281,Z 687.896,A -85,B 0,C 180,E1 -17986.363,E2 -17986.363} C_VEL
LIN {X 0,Y 268.913,Z 686.552,A -85,B 0,C 180,E1 -17989.458,E2 -17989.458} C_VEL
LIN {X 0,Y 269.731,Z 684.684,A -85,B 0,C 180,E1 -17991.757,E2 -17991.757} C_VEL
LIN {X 0,Y 269.611,Z 683.527,A -85,B 0,C 180,E1 -17992.987,E2 -17992.987} C_VEL
LIN {X 0,Y 267.774,Z 681.476,A -85,B 0,C 180,E1 -17995.02,E2 -17995.02} C_VEL
LIN {X 0,Y 266.344,Z 679.512,A -85,B 0,C 180,E1 -17996.647,E2 -17996.647} C_VEL
LIN {X 0,Y 266.175,Z 677.739,A -85,B 0,C 180,E1 -17997.86,E2 -17997.86} C_VEL
LIN {X 0,Y 266.406,Z 677.033,A -85,B 0,C 180,E1 -17998.255,E2 -17998.255} C_VEL
LIN {X 0,Y 269.357,Z 670.427,A -85,B 0,C 180,E1 -18001.495,E2 -18001.495} C_VEL
LIN {X 0,Y 272.764,Z 662.645,A -85,B 0,C 180,E1 -18004.433,E2 -18004.433} C_VEL
LIN {X 0,Y 276.22,Z 654.738,A -85,B 0,C 180,E1 -18006.861,E2 -18006.861} C_VEL
LIN {X 0,Y 280.387,Z 644.646,A -85,B 0,C 180,E1 -18009.376,E2 -18009.376} C_VEL
LIN {X 0,Y 284.96,Z 632.925,A -85,B 0,C 180,E1 -18011.74,E2 -18011.74} C_VEL
LIN {X 0,Y 289.441,Z 620.497,A -85,B 0,C 180,E1 -18013.766,E2 -18013.766} C_VEL
LIN {X 0,Y 293.992,Z 606.532,A -85,B 0,C 180,E1 -18015.601,E2 -18015.601} C_VEL
LIN {X 0,Y 298.161,Z 592.031,A -85,B 0,C 180,E1 -18017.136,E2 -18017.136} C_VEL
LIN {X 0,Y 301.766,Z 577.555,A -85,B 0,C 180,E1 -18018.325,E2 -18018.325} C_VEL
LIN {X 0,Y 305.004,Z 561.646,A -85,B 0,C 180,E1 -18019.344,E2 -18019.344} C_VEL
LIN {X 0,Y 307.57,Z 545.679,A -85,B 0,C 180,E1 -18020.091,E2 -18020.091} C_VEL
LIN {X 0,Y 318.915,Z 457.071,A -85,B 0,C 180,E1 -18023.103,E2 -18023.103} C_VEL
LIN {X 0,Y 316.548,Z 451.501,A -85,B 0,C 180,E1 -18024.534,E2 -18024.534} C_VEL
LIN {X 0,Y 314.193,Z 446.827,A -85,B 0,C 180,E1 -18026.111,E2 -18026.111} C_VEL
LIN {X 0,Y 311.606,Z 441.927,A -85,B 0,C 180,E1 -18028.27,E2 -18028.27} C_VEL
LIN {X 0,Y 309.277,Z 438.185,A -85,B 0,C 180,E1 -18030.971,E2 -18030.971} C_VEL
LIN {X 0,Y 308.146,Z 436.753,A -85,B 0,C 180,E1 -18033.187,E2 -18033.187} C_VEL
LIN {X 0,Y 307.773,Z 436.59,A -85,B 0,C 180,E1 -18035.54,E2 -18035.54} C_VEL
LIN {X 0,Y 308.236,Z 438.12,A -85,B 0,C 180,E1 -18037.997,E2 -18037.997} C_VEL
LIN {X 0,Y 309.774,Z 441.084,A -85,B 0,C 180,E1 -18040.628,E2 -18040.628} C_VEL
LIN {X 0,Y 312.047,Z 446.372,A -85,B 0,C 180,E1 -18043.131,E2 -18043.131} C_VEL
LIN {X 0,Y 314.097,Z 451.352,A -85,B 0,C 180,E1 -18044.829,E2 -18044.829} C_VEL
LIN {X 0,Y 316.306,Z 456.831,A -85,B 0,C 180,E1 -18046.345,E2 -18046.345} C_VEL
LIN {X 0,Y 318.409,Z 463.067,A -85,B 0,C 180,E1 -18047.69,E2 -18047.69} C_VEL
LIN {X 0,Y 308.176,Z 544.821,A -85,B 0,C 180,E1 -18050.474,E2 -18050.474} C_VEL
LIN {X 0,Y 305.602,Z 562.675,A -85,B 0,C 180,E1 -18051.14,E2 -18051.14} C_VEL
LIN {X 0,Y 302.216,Z 580.025,A -85,B 0,C 180,E1 -18052.061,E2 -18052.061} C_VEL
LIN {X 0,Y 298.532,Z 595.113,A -85,B 0,C 180,E1 -18053.106,E2 -18053.106} C_VEL
LIN {X 0,Y 294.384,Z 609.888,A -85,B 0,C 180,E1 -18054.449,E2 -18054.449} C_VEL
LIN {X 0,Y 289.431,Z 625.511,A -85,B 0,C 180,E1 -18056.256,E2 -18056.256} C_VEL
LIN {X 0,Y 284.883,Z 638.663,A -85,B 0,C 180,E1 -18058.174,E2 -18058.174} C_VEL
LIN {X 0,Y 281.092,Z 648.862,A -85,B 0,C 180,E1 -18059.995,E2 -18059.995} C_VEL
LIN {X 0,Y 277.317,Z 658.608,A -85,B 0,C 180,E1 -18062.039,E2 -18062.039} C_VEL
LIN {X 0,Y 273.371,Z 668.284,A -85,B 0,C 180,E1 -18064.491,E2 -18064.491} C_VEL
LIN {X 0,Y 269.706,Z 677.504,A -85,B 0,C 180,E1 -18067.394,E2 -18067.394} C_VEL
LIN {X 0,Y 267.049,Z 684.235,A -85,B 0,C 180,E1 -18069.991,E2 -18069.991} C_VEL
LIN {X 0,Y 264.373,Z 690.738,A -85,B 0,C 180,E1 -18073.138,E2 -18073.138} C_VEL
LIN {X 0,Y 262.914,Z 695.404,A -85,B 0,C 180,E1 -18076.077,E2 -18076.077} C_VEL
LIN {X 0,Y 261.775,Z 699,A -85,B 0,C 180,E1 -18079.166,E2 -18079.166} C_VEL
LIN {X 0,Y 261.188,Z 701.387,A -85,B 0,C 180,E1 -18082.266,E2 -18082.266} C_VEL
LIN {X 0,Y 261.017,Z 702.581,A -85,B 0,C 180,E1 -18085.365,E2 -18085.365} C_VEL
LIN {X 0,Y 261.11,Z 702.569,A -85,B 0,C 180,E1 -18088.455,E2 -18088.455} C_VEL
LIN {X 0,Y 261.135,Z 701.303,A -85,B 0,C 180,E1 -18091.54,E2 -18091.54} C_VEL
LIN {X 0,Y 261.144,Z 700.173,A -85,B 0,C 180,E1 -18093.083,E2 -18093.083} C_VEL
LIN {X 0,Y 261.156,Z 696.877,A -85,B 0,C 180,E1 -18096.177,E2 -18096.177} C_VEL
LIN {X 0,Y 261.403,Z 692.16,A -85,B 0,C 180,E1 -18099.281,E2 -18099.281} C_VEL
LIN {X 0,Y 262.008,Z 685.896,A -85,B 0,C 180,E1 -18102.389,E2 -18102.389} C_VEL
LIN {X 0,Y 262.872,Z 678.981,A -85,B 0,C 180,E1 -18105.107,E2 -18105.107} C_VEL
LIN {X 0,Y 264.269,Z 670.603,A -85,B 0,C 180,E1 -18107.806,E2 -18107.806} C_VEL
LIN {X 0,Y 266.084,Z 660.479,A -85,B 0,C 180,E1 -18110.483,E2 -18110.483} C_VEL
LIN {X 0,Y 267.982,Z 650.079,A -85,B 0,C 180,E1 -18112.755,E2 -18112.755} C_VEL
LIN {X 0,Y 270.005,Z 638.806,A -85,B 0,C 180,E1 -18114.814,E2 -18114.814} C_VEL
LIN {X 0,Y 272.169,Z 626.693,A -85,B 0,C 180,E1 -18116.655,E2 -18116.655} C_VEL
LIN {X 0,Y 274.316,Z 613.678,A -85,B 0,C 180,E1 -18118.29,E2 -18118.29} C_VEL
LIN {X 0,Y 276.526,Z 599.708,A -85,B 0,C 180,E1 -18119.706,E2 -18119.706} C_VEL
LIN {X 0,Y 278.431,Z 584.667,A -85,B 0,C 180,E1 -18120.919,E2 -18120.919} C_VEL
LIN {X 0,Y 280.067,Z 569.294,A -85,B 0,C 180,E1 -18121.851,E2 -18121.851} C_VEL
LIN {X 0,Y 281.288,Z 554.43,A -85,B 0,C 180,E1 -18122.489,E2 -18122.489} C_VEL
LIN {X 0,Y 287.307,Z 448.642,A -85,B 0,C 180,E1 -18125.902,E2 -18125.902} C_VEL
LIN {X 0,Y 285.844,Z 440.325,A -85,B 0,C 180,E1 -18126.36,E2 -18126.36} C_VEL
LIN {X 0,Y 275.007,Z 413.401,A -85,B 0,C 180,E1 -18128.579,E2 -18128.579} C_VEL
LIN {X 0,Y 266.945,Z 395.196,A -85,B 0,C 180,E1 -18130.3,E2 -18130.3} C_VEL
LIN {X 0,Y 265.605,Z 392.042,A -85,B 0,C 180,E1 -18130.615,E2 -18130.615} C_VEL
LIN {X 0,Y 263.069,Z 382.342,A -85,B 0,C 180,E1 -18133.837,E2 -18133.837} C_VEL
LIN {X 0,Y 263.098,Z 382.34,A -85,B 0,C 180,E1 -18138.409,E2 -18138.409} C_VEL
LIN {X 0,Y 263.136,Z 382.337,A -85,B 0,C 180,E1 -18142.099,E2 -18142.099} C_VEL
LIN {X 0,Y 263.14,Z 382.334,A -85,B 0,C 180,E1 -18145.884,E2 -18145.884} C_VEL
LIN {X 0,Y 263.096,Z 382.337,A -85,B 0,C 180,E1 -18149.5,E2 -18149.5} C_VEL
LIN {X 0,Y 263.099,Z 382.334,A -85,B 0,C 180,E1 -18152.993,E2 -18152.993} C_VEL
LIN {X 0,Y 263.104,Z 382.338,A -85,B 0,C 180,E1 -18156.38,E2 -18156.38} C_VEL
LIN {X 0,Y 263.195,Z 382.325,A -85,B 0,C 180,E1 -18159.688,E2 -18159.688} C_VEL
LIN {X 0,Y 263.282,Z 382.314,A -85,B 0,C 180,E1 -18164.518,E2 -18164.518} C_VEL
LIN {X 0,Y 263.316,Z 382.3,A -85,B 0,C 180,E1 -18169.232,E2 -18169.232} C_VEL
LIN {X 0,Y 263.512,Z 382.285,A -85,B 0,C 180,E1 -18172.337,E2 -18172.337} C_VEL
LIN {X 0,Y 263.719,Z 382.259,A -85,B 0,C 180,E1 -18178.473,E2 -18178.473} C_VEL
LIN {X 0,Y 263.719,Z 382.259,A -85,B 0,C 180,E1 -18181.528,E2 -18181.528} C_VEL
LIN {X 0,Y 263.513,Z 382.286,A -85,B 0,C 180,E1 -18187.664,E2 -18187.664} C_VEL
LIN {X 0,Y 263.316,Z 382.305,A -85,B 0,C 180,E1 -18190.768,E2 -18190.768} C_VEL
LIN {X 0,Y 263.283,Z 382.313,A -85,B 0,C 180,E1 -18195.483,E2 -18195.483} C_VEL
LIN {X 0,Y 263.196,Z 382.325,A -85,B 0,C 180,E1 -18200.313,E2 -18200.313} C_VEL
LIN {X 0,Y 263.11,Z 382.33,A -85,B 0,C 180,E1 -18205.302,E2 -18205.302} C_VEL
LIN {X 0,Y 263.107,Z 382.334,A -85,B 0,C 180,E1 -18208.739,E2 -18208.739} C_VEL
LIN {X 0,Y 263.116,Z 382.331,A -85,B 0,C 180,E1 -18212.291,E2 -18212.291} C_VEL
LIN {X 0,Y 263.164,Z 382.326,A -85,B 0,C 180,E1 -18216.763,E2 -18216.763} C_VEL
LIN {X 0,Y 263.082,Z 382.339,A -85,B 0,C 180,E1 -18219.877,E2 -18219.877} C_VEL
LIN {X 0,Y 263.068,Z 382.34,A -85,B 0,C 180,E1 -18223.996,E2 -18223.996} C_VEL
LIN {X 0,Y 263.068,Z 382.34,A -85,B 0,C 180,E1 -18228.099,E2 -18228.099} C_VEL
LIN {X 0,Y 263.097,Z 382.336,A -85,B 0,C 180,E1 -18232.096,E2 -18232.096} C_VEL
LIN {X 0,Y 263.147,Z 382.332,A -85,B 0,C 180,E1 -18235.888,E2 -18235.888} C_VEL
LIN {X 0,Y 263.105,Z 382.333,A -85,B 0,C 180,E1 -18239.504,E2 -18239.504} C_VEL
LIN {X 0,Y 263.11,Z 382.334,A -85,B 0,C 180,E1 -18242.996,E2 -18242.996} C_VEL
LIN {X 0,Y 263.122,Z 382.331,A -85,B 0,C 180,E1 -18246.384,E2 -18246.384} C_VEL
LIN {X 0,Y 263.236,Z 382.322,A -85,B 0,C 180,E1 -18249.694,E2 -18249.694} C_VEL
LIN {X 0,Y 263.323,Z 382.292,A -85,B 0,C 180,E1 -18254.523,E2 -18254.523} C_VEL
LIN {X 0,Y 263.355,Z 382.303,A -85,B 0,C 180,E1 -18259.236,E2 -18259.236} C_VEL
LIN {X 0,Y 263.527,Z 382.28,A -85,B 0,C 180,E1 -18262.339,E2 -18262.339} C_VEL
LIN {X 0,Y 263.741,Z 382.256,A -85,B 0,C 180,E1 -18268.475,E2 -18268.475} C_VEL
LIN {X 0,Y 263.737,Z 382.256,A -85,B 0,C 180,E1 -18271.529,E2 -18271.529} C_VEL
LIN {X 0,Y 263.534,Z 382.283,A -85,B 0,C 180,E1 -18277.665,E2 -18277.665} C_VEL
LIN {X 0,Y 263.352,Z 382.303,A -85,B 0,C 180,E1 -18280.769,E2 -18280.769} C_VEL
LIN {X 0,Y 263.293,Z 382.312,A -85,B 0,C 180,E1 -18285.484,E2 -18285.484} C_VEL
LIN {X 0,Y 263.241,Z 382.319,A -85,B 0,C 180,E1 -18290.311,E2 -18290.311} C_VEL
LIN {X 0,Y 263.143,Z 382.33,A -85,B 0,C 180,E1 -18295.3,E2 -18295.3} C_VEL
LIN {X 0,Y 263.143,Z 382.332,A -85,B 0,C 180,E1 -18299.612,E2 -18299.612} C_VEL
LIN {X 0,Y 263.143,Z 382.333,A -85,B 0,C 180,E1 -18300.385,E2 -18300.385} C_VEL
LIN {X 0,Y 264.248,Z 385.33,A -85,B 0,C 180,E1 -18300.679,E2 -18300.679} C_VEL
LIN {X 0,Y 274.662,Z 405.474,A -85,B 0,C 180,E1 -18302.772,E2 -18302.772} C_VEL
LIN {X 0,Y 283.861,Z 426.814,A -85,B 0,C 180,E1 -18304.627,E2 -18304.627} C_VEL
LIN {X 0,Y 287.414,Z 435.953,A -85,B 0,C 180,E1 -18305.333,E2 -18305.333} C_VEL
LIN {X 0,Y 281.12,Z 543.848,A -85,B 0,C 180,E1 -18308.815,E2 -18308.815} C_VEL
LIN {X 0,Y 279.796,Z 559.198,A -85,B 0,C 180,E1 -18309.572,E2 -18309.572} C_VEL
LIN {X 0,Y 278.21,Z 574.16,A -85,B 0,C 180,E1 -18310.586,E2 -18310.586} C_VEL
LIN {X 0,Y 276.462,Z 587.835,A -85,B 0,C 180,E1 -18311.771,E2 -18311.771} C_VEL
LIN {X 0,Y 274.427,Z 601.409,A -85,B 0,C 180,E1 -18313.23,E2 -18313.23} C_VEL
LIN {X 0,Y 272.214,Z 614.984,A -85,B 0,C 180,E1 -18315.027,E2 -18315.027} C_VEL
LIN {X 0,Y 269.979,Z 627.46,A -85,B 0,C 180,E1 -18317.036,E2 -18317.036} C_VEL
LIN {X 0,Y 268.086,Z 637.909,A -85,B 0,C 180,E1 -18319.05,E2 -18319.05} C_VEL
LIN {X 0,Y 266.05,Z 649.04,A -85,B 0,C 180,E1 -18321.626,E2 -18321.626} C_VEL
LIN {X 0,Y 264.436,Z 658.256,A -85,B 0,C 180,E1 -18324.217,E2 -18324.217} C_VEL
LIN {X 0,Y 263.001,Z 667,A -85,B 0,C 180,E1 -18327.239,E2 -18327.239} C_VEL
LIN {X 0,Y 262.052,Z 673.974,A -85,B 0,C 180,E1 -18330.254,E2 -18330.254} C_VEL
LIN {X 0,Y 261.51,Z 678.698,A -85,B 0,C 180,E1 -18332.814,E2 -18332.814} C_VEL
LIN {X 0,Y 261.046,Z 682.337,A -85,B 0,C 180,E1 -18335.335,E2 -18335.335} C_VEL
LIN {X 0,Y 260.797,Z 685.1,A -85,B 0,C 180,E1 -18337.835,E2 -18337.835} C_VEL
LIN {X 0,Y 260.756,Z 687.419,A -85,B 0,C 180,E1 -18341.129,E2 -18341.129} C_VEL
LIN {X 0,Y 260.879,Z 688.332,A -85,B 0,C 180,E1 -18344.371,E2 -18344.371} C_VEL
LIN {X 0,Y 261.372,Z 687.924,A -85,B 0,C 180,E1 -18347.578,E2 -18347.578} C_VEL
LIN {X 0,Y 262.247,Z 686.264,A -85,B 0,C 180,E1 -18350.746,E2 -18350.746} C_VEL
LIN {X 0,Y 263.565,Z 683.37,A -85,B 0,C 180,E1 -18353.877,E2 -18353.877} C_VEL
LIN {X 0,Y 265.44,Z 679.189,A -85,B 0,C 180,E1 -18356.964,E2 -18356.964} C_VEL
LIN {X 0,Y 266.406,Z 677.033,A -85,B 0,C 180,E1 -18358.255,E2 -18358.255} C_VEL
LIN {X 0,Y 266.746,Z 675.022,A -85,B 0,C 180,E1 -18359.445,E2 -18359.445} C_VEL
LIN {X 0,Y 265.75,Z 671.68,A -85,B 0,C 180,E1 -18361.444,E2 -18361.444} C_VEL
LIN {X 0,Y 265.02,Z 667.985,A -85,B 0,C 180,E1 -18363.42,E2 -18363.42} C_VEL
LIN {X 0,Y 265.756,Z 665.296,A -85,B 0,C 180,E1 -18364.546,E2 -18364.546} C_VEL
LIN {X 0,Y 269.954,Z 656.322,A -85,B 0,C 180,E1 -18367.479,E2 -18367.479} C_VEL
LIN {X 0,Y 274.188,Z 646.878,A -85,B 0,C 180,E1 -18369.963,E2 -18369.963} C_VEL
LIN {X 0,Y 278.967,Z 635.594,A -85,B 0,C 180,E1 -18372.365,E2 -18372.365} C_VEL
LIN {X 0,Y 284.243,Z 621.894,A -85,B 0,C 180,E1 -18374.691,E2 -18374.691} C_VEL
LIN {X 0,Y 288.769,Z 609.072,A -85,B 0,C 180,E1 -18376.435,E2 -18376.435} C_VEL
LIN {X 0,Y 293.068,Z 595.043,A -85,B 0,C 180,E1 -18377.984,E2 -18377.984} C_VEL
LIN {X 0,Y 296.81,Z 581.427,A -85,B 0,C 180,E1 -18379.18,E2 -18379.18} C_VEL
LIN {X 0,Y 300.094,Z 567.073,A -85,B 0,C 180,E1 -18380.18,E2 -18380.18} C_VEL
LIN {X 0,Y 302.959,Z 551.691,A -85,B 0,C 180,E1 -18380.976,E2 -18380.976} C_VEL
LIN {X 0,Y 306.095,Z 529.055,A -85,B 0,C 180,E1 -18381.818,E2 -18381.818} C_VEL
LIN {X 0,Y 315.364,Z 460.763,A -85,B 0,C 180,E1 -18384.159,E2 -18384.159} C_VEL
LIN {X 0,Y 312.867,Z 454.859,A -85,B 0,C 180,E1 -18385.887,E2 -18385.887} C_VEL
LIN {X 0,Y 310.802,Z 450.863,A -85,B 0,C 180,E1 -18387.51,E2 -18387.51} C_VEL
LIN {X 0,Y 309.377,Z 448.008,A -85,B 0,C 180,E1 -18388.937,E2 -18388.937} C_VEL
LIN {X 0,Y 307.651,Z 445.016,A -85,B 0,C 180,E1 -18391.158,E2 -18391.158} C_VEL
LIN {X 0,Y 306.604,Z 443.618,A -85,B 0,C 180,E1 -18393.376,E2 -18393.376} C_VEL
LIN {X 0,Y 306.32,Z 443.596,A -85,B 0,C 180,E1 -18395.735,E2 -18395.735} C_VEL
LIN {X 0,Y 306.89,Z 445.495,A -85,B 0,C 180,E1 -18398.362,E2 -18398.362} C_VEL
LIN {X 0,Y 308.069,Z 447.926,A -85,B 0,C 180,E1 -18400.39,E2 -18400.39} C_VEL
LIN {X 0,Y 309.99,Z 452.756,A -85,B 0,C 180,E1 -18402.69,E2 -18402.69} C_VEL
LIN {X 0,Y 311.686,Z 457.138,A -85,B 0,C 180,E1 -18404.224,E2 -18404.224} C_VEL
LIN {X 0,Y 313.536,Z 462.211,A -85,B 0,C 180,E1 -18405.663,E2 -18405.663} C_VEL
LIN {X 0,Y 314.868,Z 466.712,A -85,B 0,C 180,E1 -18406.665,E2 -18406.665} C_VEL
LIN {X 0,Y 302.564,Z 557.951,A -85,B 0,C 180,E1 -18409.809,E2 -18409.809} C_VEL
LIN {X 0,Y 299.548,Z 573.984,A -85,B 0,C 180,E1 -18410.582,E2 -18410.582} C_VEL
LIN {X 0,Y 295.648,Z 590.071,A -85,B 0,C 180,E1 -18411.607,E2 -18411.607} C_VEL
LIN {X 0,Y 291.297,Z 605.379,A -85,B 0,C 180,E1 -18412.901,E2 -18412.901} C_VEL
LIN {X 0,Y 287.223,Z 618.12,A -85,B 0,C 180,E1 -18414.252,E2 -18414.252} C_VEL
LIN {X 0,Y 282.542,Z 631.235,A -85,B 0,C 180,E1 -18415.965,E2 -18415.965} C_VEL
LIN {X 0,Y 277.885,Z 643.373,A -85,B 0,C 180,E1 -18417.917,E2 -18417.917} C_VEL
LIN {X 0,Y 273.737,Z 653.732,A -85,B 0,C 180,E1 -18419.955,E2 -18419.955} C_VEL
LIN {X 0,Y 269.346,Z 664.051,A -85,B 0,C 180,E1 -18422.41,E2 -18422.41} C_VEL
LIN {X 0,Y 265.512,Z 672.824,A -85,B 0,C 180,E1 -18424.941,E2 -18424.941} C_VEL
LIN {X 0,Y 261.972,Z 681.132,A -85,B 0,C 180,E1 -18427.938,E2 -18427.938} C_VEL
LIN {X 0,Y 258.981,Z 687.958,A -85,B 0,C 180,E1 -18430.993,E2 -18430.993} C_VEL
LIN {X 0,Y 256.699,Z 693.368,A -85,B 0,C 180,E1 -18434.108,E2 -18434.108} C_VEL
LIN {X 0,Y 255.248,Z 697.496,A -85,B 0,C 180,E1 -18437.273,E2 -18437.273} C_VEL
LIN {X 0,Y 254.38,Z 700.357,A -85,B 0,C 180,E1 -18440.456,E2 -18440.456} C_VEL
LIN {X 0,Y 253.962,Z 702.008,A -85,B 0,C 180,E1 -18443.642,E2 -18443.642} C_VEL
LIN {X 0,Y 253.953,Z 702.477,A -85,B 0,C 180,E1 -18446.825,E2 -18446.825} C_VEL
LIN {X 0,Y 254.038,Z 702.255,A -85,B 0,C 180,E1 -18448.412,E2 -18448.412} C_VEL
LIN {X 0,Y 254.064,Z 700.863,A -85,B 0,C 180,E1 -18451.583,E2 -18451.583} C_VEL
LIN {X 0,Y 254.059,Z 698.162,A -85,B 0,C 180,E1 -18454.758,E2 -18454.758} C_VEL
LIN {X 0,Y 254.207,Z 694.069,A -85,B 0,C 180,E1 -18457.943,E2 -18457.943} C_VEL
LIN {X 0,Y 254.586,Z 688.459,A -85,B 0,C 180,E1 -18461.139,E2 -18461.139} C_VEL
LIN {X 0,Y 255.266,Z 683.145,A -85,B 0,C 180,E1 -18463.531,E2 -18463.531} C_VEL
LIN {X 0,Y 256.391,Z 675.486,A -85,B 0,C 180,E1 -18466.385,E2 -18466.385} C_VEL
LIN {X 0,Y 257.878,Z 666.638,A -85,B 0,C 180,E1 -18469.086,E2 -18469.086} C_VEL
LIN {X 0,Y 259.952,Z 655.712,A -85,B 0,C 180,E1 -18471.82,E2 -18471.82} C_VEL
LIN {X 0,Y 261.812,Z 645.223,A -85,B 0,C 180,E1 -18473.997,E2 -18473.997} C_VEL
LIN {X 0,Y 264.108,Z 633.382,A -85,B 0,C 180,E1 -18476.042,E2 -18476.042} C_VEL
LIN {X 0,Y 266.425,Z 620.24,A -85,B 0,C 180,E1 -18477.916,E2 -18477.916} C_VEL
LIN {X 0,Y 268.772,Z 605.911,A -85,B 0,C 180,E1 -18479.571,E2 -18479.571} C_VEL
LIN {X 0,Y 270.94,Z 591.154,A -85,B 0,C 180,E1 -18480.922,E2 -18480.922} C_VEL
LIN {X 0,Y 272.783,Z 576.096,A -85,B 0,C 180,E1 -18481.986,E2 -18481.986} C_VEL
LIN {X 0,Y 274.332,Z 559.962,A -85,B 0,C 180,E1 -18482.816,E2 -18482.816} C_VEL
LIN {X 0,Y 280.848,Z 451.822,A -85,B 0,C 180,E1 -18486.416,E2 -18486.416} C_VEL
LIN {X 0,Y 280.63,Z 448.004,A -85,B 0,C 180,E1 -18486.587,E2 -18486.587} C_VEL
LIN {X 0,Y 279.645,Z 442.705,A -85,B 0,C 180,E1 -18486.898,E2 -18486.898} C_VEL
LIN {X 0,Y 269.13,Z 416.371,A -85,B 0,C 180,E1 -18489.145,E2 -18489.145} C_VEL
LIN {X 0,Y 260.927,Z 397.906,A -85,B 0,C 180,E1 -18490.928,E2 -18490.928} C_VEL
LIN {X 0,Y 258.291,Z 391.842,A -85,B 0,C 180,E1 -18491.56,E2 -18491.56} C_VEL
LIN {X 0,Y 255.99,Z 383.224,A -85,B 0,C 180,E1 -18494.531,E2 -18494.531} C_VEL
LIN {X 0,Y 256.028,Z 383.219,A -85,B 0,C 180,E1 -18498.792,E2 -18498.792} C_VEL
LIN {X 0,Y 256.109,Z 383.209,A -85,B 0,C 180,E1 -18502.864,E2 -18502.864} C_VEL
LIN {X 0,Y 256.053,Z 383.215,A -85,B 0,C 180,E1 -18506.706,E2 -18506.706} C_VEL
LIN {X 0,Y 256.028,Z 383.219,A -85,B 0,C 180,E1 -18510.39,E2 -18510.39} C_VEL
LIN {X 0,Y 256.053,Z 383.211,A -85,B 0,C 180,E1 -18513.95,E2 -18513.95} C_VEL
LIN {X 0,Y 256.045,Z 383.215,A -85,B 0,C 180,E1 -18517.402,E2 -18517.402} C_VEL
LIN {X 0,Y 256.096,Z 383.2,A -85,B 0,C 180,E1 -18520.773,E2 -18520.773} C_VEL
LIN {X 0,Y 256.207,Z 383.197,A -85,B 0,C 180,E1 -18524.08,E2 -18524.08} C_VEL
LIN {X 0,Y 256.26,Z 383.178,A -85,B 0,C 180,E1 -18528.932,E2 -18528.932} C_VEL
LIN {X 0,Y 256.455,Z 383.163,A -85,B 0,C 180,E1 -18532.125,E2 -18532.125} C_VEL
LIN {X 0,Y 256.436,Z 383.162,A -85,B 0,C 180,E1 -18536.858,E2 -18536.858} C_VEL
LIN {X 0,Y 256.681,Z 383.136,A -85,B 0,C 180,E1 -18538.431,E2 -18538.431} C_VEL
LIN {X 0,Y 256.681,Z 383.136,A -85,B 0,C 180,E1 -18541.569,E2 -18541.569} C_VEL
LIN {X 0,Y 256.432,Z 383.166,A -85,B 0,C 180,E1 -18546.577,E2 -18546.577} C_VEL
LIN {X 0,Y 256.389,Z 383.17,A -85,B 0,C 180,E1 -18549.467,E2 -18549.467} C_VEL
LIN {X 0,Y 256.192,Z 383.197,A -85,B 0,C 180,E1 -18554.294,E2 -18554.294} C_VEL
LIN {X 0,Y 256.138,Z 383.2,A -85,B 0,C 180,E1 -18557.568,E2 -18557.568} C_VEL
LIN {X 0,Y 256.107,Z 383.206,A -85,B 0,C 180,E1 -18561.099,E2 -18561.099} C_VEL
LIN {X 0,Y 256.072,Z 383.206,A -85,B 0,C 180,E1 -18565.089,E2 -18565.089} C_VEL
LIN {X 0,Y 256.065,Z 383.211,A -85,B 0,C 180,E1 -18568.571,E2 -18568.571} C_VEL
LIN {X 0,Y 256.06,Z 383.215,A -85,B 0,C 180,E1 -18571.702,E2 -18571.702} C_VEL
LIN {X 0,Y 256.069,Z 383.206,A -85,B 0,C 180,E1 -18575.195,E2 -18575.195} C_VEL
LIN {X 0,Y 256.095,Z 383.207,A -85,B 0,C 180,E1 -18577.27,E2 -18577.27} C_VEL
LIN {X 0,Y 256.031,Z 383.213,A -85,B 0,C 180,E1 -18581.209,E2 -18581.209} C_VEL
LIN {X 0,Y 256.01,Z 383.219,A -85,B 0,C 180,E1 -18585.542,E2 -18585.542} C_VEL
LIN {X 0,Y 256.002,Z 383.217,A -85,B 0,C 180,E1 -18588.79,E2 -18588.79} C_VEL
LIN {X 0,Y 256.093,Z 383.206,A -85,B 0,C 180,E1 -18592.865,E2 -18592.865} C_VEL
LIN {X 0,Y 256.061,Z 383.21,A -85,B 0,C 180,E1 -18596.709,E2 -18596.709} C_VEL
LIN {X 0,Y 256.036,Z 383.215,A -85,B 0,C 180,E1 -18600.394,E2 -18600.394} C_VEL
LIN {X 0,Y 256.065,Z 383.212,A -85,B 0,C 180,E1 -18603.954,E2 -18603.954} C_VEL
LIN {X 0,Y 256.065,Z 383.212,A -85,B 0,C 180,E1 -18607.406,E2 -18607.406} C_VEL
LIN {X 0,Y 256.157,Z 383.199,A -85,B 0,C 180,E1 -18610.78,E2 -18610.78} C_VEL
LIN {X 0,Y 256.245,Z 383.175,A -85,B 0,C 180,E1 -18614.084,E2 -18614.084} C_VEL
LIN {X 0,Y 256.29,Z 383.178,A -85,B 0,C 180,E1 -18617.33,E2 -18617.33} C_VEL
LIN {X 0,Y 256.435,Z 383.165,A -85,B 0,C 180,E1 -18620.625,E2 -18620.625} C_VEL
LIN {X 0,Y 256.456,Z 383.157,A -85,B 0,C 180,E1 -18623.709,E2 -18623.709} C_VEL
LIN {X 0,Y 256.702,Z 383.133,A -85,B 0,C 180,E1 -18628.434,E2 -18628.434} C_VEL
LIN {X 0,Y 256.7,Z 383.132,A -85,B 0,C 180,E1 -18631.571,E2 -18631.571} C_VEL
LIN {X 0,Y 256.461,Z 383.165,A -85,B 0,C 180,E1 -18636.295,E2 -18636.295} C_VEL
LIN {X 0,Y 256.432,Z 383.164,A -85,B 0,C 180,E1 -18639.467,E2 -18639.467} C_VEL
LIN {X 0,Y 256.212,Z 383.191,A -85,B 0,C 180,E1 -18644.295,E2 -18644.295} C_VEL
LIN {X 0,Y 256.166,Z 383.2,A -85,B 0,C 180,E1 -18647.567,E2 -18647.567} C_VEL
LIN {X 0,Y 256.148,Z 383.204,A -85,B 0,C 180,E1 -18651.112,E2 -18651.112} C_VEL
LIN {X 0,Y 256.112,Z 383.206,A -85,B 0,C 180,E1 -18655.1,E2 -18655.1} C_VEL
LIN {X 0,Y 256.103,Z 383.209,A -85,B 0,C 180,E1 -18659.522,E2 -18659.522} C_VEL
LIN {X 0,Y 257.176,Z 386.175,A -85,B 0,C 180,E1 -18659.805,E2 -18659.805} C_VEL
LIN {X 0,Y 267.379,Z 405.798,A -85,B 0,C 180,E1 -18661.938,E2 -18661.938} C_VEL
LIN {X 0,Y 272.101,Z 415.906,A -85,B 0,C 180,E1 -18662.904,E2 -18662.904} C_VEL
LIN {X 0,Y 280.943,Z 437.422,A -85,B 0,C 180,E1 -18664.733,E2 -18664.733} C_VEL
LIN {X 0,Y 274.515,Z 544.523,A -85,B 0,C 180,E1 -18668.293,E2 -18668.293} C_VEL
LIN {X 0,Y 273.173,Z 559.409,A -85,B 0,C 180,E1 -18669.045,E2 -18669.045} C_VEL
LIN {X 0,Y 271.46,Z 575.009,A -85,B 0,C 180,E1 -18670.136,E2 -18670.136} C_VEL
LIN {X 0,Y 269.54,Z 589.444,A -85,B 0,C 180,E1 -18671.441,E2 -18671.441} C_VEL
LIN {X 0,Y 267.403,Z 603.157,A -85,B 0,C 180,E1 -18672.984,E2 -18672.984} C_VEL
LIN {X 0,Y 265.134,Z 616.539,A -85,B 0,C 180,E1 -18674.836,E2 -18674.836} C_VEL
LIN {X 0,Y 262.806,Z 629.366,A -85,B 0,C 180,E1 -18677.005,E2 -18677.005} C_VEL
LIN {X 0,Y 260.648,Z 640.544,A -85,B 0,C 180,E1 -18679.286,E2 -18679.286} C_VEL
LIN {X 0,Y 258.628,Z 651.516,A -85,B 0,C 180,E1 -18682.007,E2 -18682.007} C_VEL
LIN {X 0,Y 256.911,Z 661.139,A -85,B 0,C 180,E1 -18684.937,E2 -18684.937} C_VEL
LIN {X 0,Y 255.753,Z 668.291,A -85,B 0,C 180,E1 -18687.598,E2 -18687.598} C_VEL
LIN {X 0,Y 254.94,Z 674.178,A -85,B 0,C 180,E1 -18690.25,E2 -18690.25} C_VEL
LIN {X 0,Y 254.404,Z 678.958,A -85,B 0,C 180,E1 -18692.918,E2 -18692.918} C_VEL
LIN {X 0,Y 253.878,Z 683.181,A -85,B 0,C 180,E1 -18696.001,E2 -18696.001} C_VEL
LIN {X 0,Y 253.632,Z 685.991,A -85,B 0,C 180,E1 -18698.886,E2 -18698.886} C_VEL
LIN {X 0,Y 253.648,Z 687.158,A -85,B 0,C 180,E1 -18700.579,E2 -18700.579} C_VEL
LIN {X 0,Y 253.75,Z 688.435,A -85,B 0,C 180,E1 -18703.92,E2 -18703.92} C_VEL
LIN {X 0,Y 254.229,Z 688.388,A -85,B 0,C 180,E1 -18707.223,E2 -18707.223} C_VEL
LIN {X 0,Y 255.058,Z 687.091,A -85,B 0,C 180,E1 -18710.483,E2 -18710.483} C_VEL
LIN {X 0,Y 256.414,Z 684.543,A -85,B 0,C 180,E1 -18713.705,E2 -18713.705} C_VEL
LIN {X 0,Y 258.27,Z 680.745,A -85,B 0,C 180,E1 -18716.88,E2 -18716.88} C_VEL
LIN {X 0,Y 260.796,Z 675.621,A -85,B 0,C 180,E1 -18720,E2 -18720} C_VEL
LIN {X 0,Y 263.892,Z 669.118,A -85,B 0,C 180,E1 -18723.053,E2 -18723.053} C_VEL
LIN {X 0,Y 265.756,Z 665.296,A -85,B 0,C 180,E1 -18724.546,E2 -18724.546} C_VEL
LIN {X 0,Y 266.594,Z 662.531,A -85,B 0,C 180,E1 -18725.658,E2 -18725.658} C_VEL
LIN {X 0,Y 266.478,Z 658.077,A -85,B 0,C 180,E1 -18727.567,E2 -18727.567} C_VEL
LIN {X 0,Y 266.579,Z 653.181,A -85,B 0,C 180,E1 -18729.416,E2 -18729.416} C_VEL
LIN {X 0,Y 267.711,Z 649.729,A -85,B 0,C 180,E1 -18730.41,E2 -18730.41} C_VEL
LIN {X 0,Y 273.003,Z 638.191,A -85,B 0,C 180,E1 -18733.017,E2 -18733.017} C_VEL
LIN {X 0,Y 277.796,Z 626.92,A -85,B 0,C 180,E1 -18735.074,E2 -18735.074} C_VEL
LIN {X 0,Y 282.699,Z 614.104,A -85,B 0,C 180,E1 -18736.984,E2 -18736.984} C_VEL
LIN {X 0,Y 287.207,Z 601.159,A -85,B 0,C 180,E1 -18738.548,E2 -18738.548} C_VEL
LIN {X 0,Y 291.318,Z 587.591,A -85,B 0,C 180,E1 -18739.866,E2 -18739.866} C_VEL
LIN {X 0,Y 295.47,Z 571.617,A -85,B 0,C 180,E1 -18741.085,E2 -18741.085} C_VEL
LIN {X 0,Y 298.655,Z 556.711,A -85,B 0,C 180,E1 -18741.936,E2 -18741.936} C_VEL
LIN {X 0,Y 301.188,Z 540.998,A -85,B 0,C 180,E1 -18742.599,E2 -18742.599} C_VEL
LIN {X 0,Y 311.991,Z 465.322,A -85,B 0,C 180,E1 -18745.196,E2 -18745.196} C_VEL
LIN {X 0,Y 311.961,Z 464.536,A -85,B 0,C 180,E1 -18745.29,E2 -18745.29} C_VEL
LIN {X 0,Y 310.017,Z 459.802,A -85,B 0,C 180,E1 -18746.847,E2 -18746.847} C_VEL
LIN {X 0,Y 307.859,Z 455.197,A -85,B 0,C 180,E1 -18748.92,E2 -18748.92} C_VEL
LIN {X 0,Y 306.031,Z 451.86,A -85,B 0,C 180,E1 -18751.342,E2 -18751.342} C_VEL
LIN {X 0,Y 305.091,Z 450.534,A -85,B 0,C 180,E1 -18753.563,E2 -18753.563} C_VEL
LIN {X 0,Y 304.864,Z 450.635,A -85,B 0,C 180,E1 -18755.932,E2 -18755.932} C_VEL
LIN {X 0,Y 305.55,Z 452.899,A -85,B 0,C 180,E1 -18758.731,E2 -18758.731} C_VEL
LIN {X 0,Y 306.317,Z 454.627,A -85,B 0,C 180,E1 -18760.072,E2 -18760.072} C_VEL
LIN {X 0,Y 307.97,Z 459.162,A -85,B 0,C 180,E1 -18762.252,E2 -18762.252} C_VEL
LIN {X 0,Y 309.368,Z 463.168,A -85,B 0,C 180,E1 -18763.678,E2 -18763.678} C_VEL
LIN {X 0,Y 311.137,Z 468.63,A -85,B 0,C 180,E1 -18765.226,E2 -18765.226} C_VEL
LIN {X 0,Y 311.576,Z 470.248,A -85,B 0,C 180,E1 -18765.585,E2 -18765.585} C_VEL
LIN {X 0,Y 299.203,Z 557.065,A -85,B 0,C 180,E1 -18768.594,E2 -18768.594} C_VEL
LIN {X 0,Y 296.32,Z 571.77,A -85,B 0,C 180,E1 -18769.288,E2 -18769.288} C_VEL
LIN {X 0,Y 292.057,Z 588.735,A -85,B 0,C 180,E1 -18770.345,E2 -18770.345} C_VEL
LIN {X 0,Y 288.133,Z 602.15,A -85,B 0,C 180,E1 -18771.431,E2 -18771.431} C_VEL
LIN {X 0,Y 283.51,Z 615.985,A -85,B 0,C 180,E1 -18772.848,E2 -18772.848} C_VEL
LIN {X 0,Y 278.15,Z 630.301,A -85,B 0,C 180,E1 -18774.689,E2 -18774.689} C_VEL
LIN {X 0,Y 272.891,Z 643.383,A -85,B 0,C 180,E1 -18776.818,E2 -18776.818} C_VEL
LIN {X 0,Y 267.75,Z 655.221,A -85,B 0,C 180,E1 -18779.211,E2 -18779.211} C_VEL
LIN {X 0,Y 263.233,Z 665.155,A -85,B 0,C 180,E1 -18781.683,E2 -18781.683} C_VEL
LIN {X 0,Y 259.141,Z 673.7,A -85,B 0,C 180,E1 -18784.281,E2 -18784.281} C_VEL
LIN {X 0,Y 255.422,Z 681.813,A -85,B 0,C 180,E1 -18787.341,E2 -18787.341} C_VEL
LIN {X 0,Y 252.25,Z 688.393,A -85,B 0,C 180,E1 -18790.466,E2 -18790.466} C_VEL
LIN {X 0,Y 249.832,Z 693.638,A -85,B 0,C 180,E1 -18793.659,E2 -18793.659} C_VEL
LIN {X 0,Y 248.285,Z 697.599,A -85,B 0,C 180,E1 -18796.91,E2 -18796.91} C_VEL
LIN {X 0,Y 247.339,Z 700.359,A -85,B 0,C 180,E1 -18800.182,E2 -18800.182} C_VEL
LIN {X 0,Y 246.879,Z 701.891,A -85,B 0,C 180,E1 -18803.459,E2 -18803.459} C_VEL
LIN {X 0,Y 246.853,Z 702.223,A -85,B 0,C 180,E1 -18806.733,E2 -18806.733} C_VEL
LIN {X 0,Y 246.965,Z 701.941,A -85,B 0,C 180,E1 -18808.367,E2 -18808.367} C_VEL
LIN {X 0,Y 246.994,Z 700.42,A -85,B 0,C 180,E1 -18811.628,E2 -18811.628} C_VEL
LIN {X 0,Y 246.988,Z 697.58,A -85,B 0,C 180,E1 -18814.894,E2 -18814.894} C_VEL
LIN {X 0,Y 247.137,Z 693.338,A -85,B 0,C 180,E1 -18818.172,E2 -18818.172} C_VEL
LIN {X 0,Y 247.557,Z 687.562,A -85,B 0,C 180,E1 -18821.46,E2 -18821.46} C_VEL
LIN {X 0,Y 248.41,Z 681.18,A -85,B 0,C 180,E1 -18824.33,E2 -18824.33} C_VEL
LIN {X 0,Y 249.607,Z 673.589,A -85,B 0,C 180,E1 -18827.109,E2 -18827.109} C_VEL
LIN {X 0,Y 251.337,Z 663.861,A -85,B 0,C 180,E1 -18830.029,E2 -18830.029} C_VEL
LIN {X 0,Y 253.245,Z 654.154,A -85,B 0,C 180,E1 -18832.429,E2 -18832.429} C_VEL
LIN {X 0,Y 255.557,Z 641.813,A -85,B 0,C 180,E1 -18834.964,E2 -18834.964} C_VEL
LIN {X 0,Y 257.836,Z 630.085,A -85,B 0,C 180,E1 -18836.944,E2 -18836.944} C_VEL
LIN {X 0,Y 260.284,Z 616.312,A -85,B 0,C 180,E1 -18838.855,E2 -18838.855} C_VEL
LIN {X 0,Y 262.494,Z 603.024,A -85,B 0,C 180,E1 -18840.352,E2 -18840.352} C_VEL
LIN {X 0,Y 264.576,Z 588.947,A -85,B 0,C 180,E1 -18841.619,E2 -18841.619} C_VEL
LIN {X 0,Y 266.524,Z 572.941,A -85,B 0,C 180,E1 -18842.719,E2 -18842.719} C_VEL
LIN {X 0,Y 268.021,Z 556.465,A -85,B 0,C 180,E1 -18843.522,E2 -18843.522} C_VEL
LIN {X 0,Y 274.54,Z 450.995,A -85,B 0,C 180,E1 -18847.105,E2 -18847.105} C_VEL
LIN {X 0,Y 273.555,Z 445.301,A -85,B 0,C 180,E1 -18847.443,E2 -18847.443} C_VEL
LIN {X 0,Y 262.959,Z 418.815,A -85,B 0,C 180,E1 -18849.754,E2 -18849.754} C_VEL
LIN {X 0,Y 255.483,Z 401.782,A -85,B 0,C 180,E1 -18851.454,E2 -18851.454} C_VEL
LIN {X 0,Y 250.945,Z 391.587,A -85,B 0,C 180,E1 -18852.569,E2 -18852.569} C_VEL
LIN {X 0,Y 248.962,Z 384.098,A -85,B 0,C 180,E1 -18855.254,E2 -18855.254} C_VEL
LIN {X 0,Y 248.975,Z 384.098,A -85,B 0,C 180,E1 -18859.649,E2 -18859.649} C_VEL
LIN {X 0,Y 249.012,Z 384.094,A -85,B 0,C 180,E1 -18863.652,E2 -18863.652} C_VEL
LIN {X 0,Y 249.019,Z 384.092,A -85,B 0,C 180,E1 -18867.847,E2 -18867.847} C_VEL
LIN {X 0,Y 249.022,Z 384.089,A -85,B 0,C 180,E1 -18871.329,E2 -18871.329} C_VEL
LIN {X 0,Y 249.043,Z 384.083,A -85,B 0,C 180,E1 -18874.957,E2 -18874.957} C_VEL
LIN {X 0,Y 249.037,Z 384.087,A -85,B 0,C 180,E1 -18878.627,E2 -18878.627} C_VEL
LIN {X 0,Y 249.145,Z 384.073,A -85,B 0,C 180,E1 -18883.616,E2 -18883.616} C_VEL
LIN {X 0,Y 249.205,Z 384.057,A -85,B 0,C 180,E1 -18888.615,E2 -18888.615} C_VEL
LIN {X 0,Y 249.401,Z 384.039,A -85,B 0,C 180,E1 -18891.901,E2 -18891.901} C_VEL
LIN {X 0,Y 249.247,Z 384.061,A -85,B 0,C 180,E1 -18895.148,E2 -18895.148} C_VEL
LIN {X 0,Y 249.643,Z 384.013,A -85,B 0,C 180,E1 -18898.387,E2 -18898.387} C_VEL
LIN {X 0,Y 249.643,Z 384.013,A -85,B 0,C 180,E1 -18901.614,E2 -18901.614} C_VEL
LIN {X 0,Y 249.41,Z 384.041,A -85,B 0,C 180,E1 -18906.558,E2 -18906.558} C_VEL
LIN {X 0,Y 249.32,Z 384.051,A -85,B 0,C 180,E1 -18909.738,E2 -18909.738} C_VEL
LIN {X 0,Y 249.138,Z 384.074,A -85,B 0,C 180,E1 -18914.708,E2 -18914.708} C_VEL
LIN {X 0,Y 249.07,Z 384.081,A -85,B 0,C 180,E1 -18918.083,E2 -18918.083} C_VEL
LIN {X 0,Y 249.031,Z 384.089,A -85,B 0,C 180,E1 -18921.524,E2 -18921.524} C_VEL
LIN {X 0,Y 249.033,Z 384.084,A -85,B 0,C 180,E1 -18925.442,E2 -18925.442} C_VEL
LIN {X 0,Y 249.013,Z 384.089,A -85,B 0,C 180,E1 -18928.97,E2 -18928.97} C_VEL
LIN {X 0,Y 249.016,Z 384.087,A -85,B 0,C 180,E1 -18932.429,E2 -18932.429} C_VEL
LIN {X 0,Y 249.014,Z 384.089,A -85,B 0,C 180,E1 -18936.349,E2 -18936.349} C_VEL
LIN {X 0,Y 248.976,Z 384.092,A -85,B 0,C 180,E1 -18940.485,E2 -18940.485} C_VEL
LIN {X 0,Y 248.975,Z 384.088,A -85,B 0,C 180,E1 -18942.788,E2 -18942.788} C_VEL
LIN {X 0,Y 248.97,Z 384.096,A -85,B 0,C 180,E1 -18947.357,E2 -18947.357} C_VEL
LIN {X 0,Y 249.015,Z 384.09,A -85,B 0,C 180,E1 -18952.21,E2 -18952.21} C_VEL
LIN {X 0,Y 249.038,Z 384.09,A -85,B 0,C 180,E1 -18955.642,E2 -18955.642} C_VEL
LIN {X 0,Y 248.989,Z 384.09,A -85,B 0,C 180,E1 -18959.468,E2 -18959.468} C_VEL
LIN {X 0,Y 249.011,Z 384.091,A -85,B 0,C 180,E1 -18963.158,E2 -18963.158} C_VEL
LIN {X 0,Y 249.011,Z 384.088,A -85,B 0,C 180,E1 -18966.729,E2 -18966.729} C_VEL
LIN {X 0,Y 249.084,Z 384.081,A -85,B 0,C 180,E1 -18970.212,E2 -18970.212} C_VEL
LIN {X 0,Y 249.196,Z 384.056,A -85,B 0,C 180,E1 -18973.621,E2 -18973.621} C_VEL
LIN {X 0,Y 249.244,Z 384.06,A -85,B 0,C 180,E1 -18978.619,E2 -18978.619} C_VEL
LIN {X 0,Y 249.419,Z 384.039,A -85,B 0,C 180,E1 -18981.903,E2 -18981.903} C_VEL
LIN {X 0,Y 249.263,Z 384.049,A -85,B 0,C 180,E1 -18985.15,E2 -18985.15} C_VEL
LIN {X 0,Y 249.663,Z 384.011,A -85,B 0,C 180,E1 -18988.389,E2 -18988.389} C_VEL
LIN {X 0,Y 249.661,Z 384.007,A -85,B 0,C 180,E1 -18991.615,E2 -18991.615} C_VEL
LIN {X 0,Y 249.433,Z 384.04,A -85,B 0,C 180,E1 -18996.474,E2 -18996.474} C_VEL
LIN {X 0,Y 249.347,Z 384.047,A -85,B 0,C 180,E1 -18999.739,E2 -18999.739} C_VEL
LIN {X 0,Y 249.155,Z 384.069,A -85,B 0,C 180,E1 -19004.709,E2 -19004.709} C_VEL
LIN {X 0,Y 249.103,Z 384.077,A -85,B 0,C 180,E1 -19008.082,E2 -19008.082} C_VEL
LIN {X 0,Y 249.086,Z 384.082,A -85,B 0,C 180,E1 -19011.52,E2 -19011.52} C_VEL
LIN {X 0,Y 249.07,Z 384.083,A -85,B 0,C 180,E1 -19015.451,E2 -19015.451} C_VEL
LIN {X 0,Y 249.068,Z 384.092,A -85,B 0,C 180,E1 -19018.61,E2 -19018.61} C_VEL
LIN {X 0,Y 249.993,Z 386.82,A -85,B 0,C 180,E1 -19018.864,E2 -19018.864} C_VEL
LIN {X 0,Y 260.585,Z 407.032,A -85,B 0,C 180,E1 -19021.171,E2 -19021.171} C_VEL
LIN {X 0,Y 265.958,Z 418.405,A -85,B 0,C 180,E1 -19022.305,E2 -19022.305} C_VEL
LIN {X 0,Y 274.439,Z 439.047,A -85,B 0,C 180,E1 -19024.109,E2 -19024.109} C_VEL
LIN {X 0,Y 271.565,Z 486.441,A -85,B 0,C 180,E1 -19025.71,E2 -19025.71} C_VEL
LIN {X 0,Y 267.961,Z 544.819,A -85,B 0,C 180,E1 -19027.727,E2 -19027.727} C_VEL
LIN {X 0,Y 266.481,Z 560.344,A -85,B 0,C 180,E1 -19028.543,E2 -19028.543} C_VEL
LIN {X 0,Y 264.757,Z 575.739,A -85,B 0,C 180,E1 -19029.663,E2 -19029.663} C_VEL
LIN {X 0,Y 262.673,Z 590.506,A -85,B 0,C 180,E1 -19031.046,E2 -19031.046} C_VEL
LIN {X 0,Y 260.366,Z 604.761,A -85,B 0,C 180,E1 -19032.721,E2 -19032.721} C_VEL
LIN {X 0,Y 258.025,Z 617.983,A -85,B 0,C 180,E1 -19034.635,E2 -19034.635} C_VEL
LIN {X 0,Y 255.711,Z 630.574,A -85,B 0,C 180,E1 -19036.86,E2 -19036.86} C_VEL
LIN {X 0,Y 253.41,Z 642.112,A -85,B 0,C 180,E1 -19039.326,E2 -19039.326} C_VEL
LIN {X 0,Y 251.442,Z 652.603,A -85,B 0,C 180,E1 -19042.053,E2 -19042.053} C_VEL
LIN {X 0,Y 249.916,Z 660.849,A -85,B 0,C 180,E1 -19044.642,E2 -19044.642} C_VEL
LIN {X 0,Y 248.659,Z 668.44,A -85,B 0,C 180,E1 -19047.519,E2 -19047.519} C_VEL
LIN {X 0,Y 247.843,Z 674.353,A -85,B 0,C 180,E1 -19050.248,E2 -19050.248} C_VEL
LIN {X 0,Y 247.311,Z 679.089,A -85,B 0,C 180,E1 -19052.955,E2 -19052.955} C_VEL
LIN {X 0,Y 246.81,Z 682.812,A -85,B 0,C 180,E1 -19055.678,E2 -19055.678} C_VEL
LIN {X 0,Y 246.566,Z 685.517,A -85,B 0,C 180,E1 -19058.25,E2 -19058.25} C_VEL
LIN {X 0,Y 246.547,Z 686.987,A -85,B 0,C 180,E1 -19060.173,E2 -19060.173} C_VEL
LIN {X 0,Y 246.618,Z 688.488,A -85,B 0,C 180,E1 -19063.442,E2 -19063.442} C_VEL
LIN {X 0,Y 247.05,Z 688.772,A -85,B 0,C 180,E1 -19066.845,E2 -19066.845} C_VEL
